// TwinCAT 3 PLC project PLC_1
// ProgramVersion: 3.1.4026.25
// libraries:
//   SPT Base Types, * (Beckhoff Automation LLC)
//   SPT Components, * (Beckhoff Automation LLC)
//   SPT Event Logger, * (Beckhoff Automation LLC)
//   Tc3_PackML_V2, * (Beckhoff Automation GmbH)
//   Tc3_EventLogger, * (Beckhoff Automation GmbH)
//   Tc2_Standard, * (Beckhoff Automation GmbH)
//   Tc2_System, * (Beckhoff Automation GmbH)
// project tree:
//   Library/DUTs/ ST_AbstractLightSource_Command.TcDUT, ST_AbstractLightSource_HMI.TcDUT, ST_AbstractLightSource_Status.TcDUT, ST_AbstractBinaryDrive_Command.TcDUT, ST_AbstractBinaryDrive_Config.TcDUT, ST_AbstractBinaryDrive_Status.TcDUT, ST_AbstractBinaryDrive_HMI.TcDUT, ST_BaseModule_HMI.TcDUT, ST_Sequence_Status.TcDUT, ST_FG_System_Safety.TcDUT, ST_IlluminatedButton_Config.TcDUT, ST_IlluminatedButton_Status.TcDUT, ST_IlluminatedButton_HMI.TcDUT, ST_SafetyDoor_Config.TcDUT, ST_SafetyDoor_Status.TcDUT, ST_SafetyDoor_HMI.TcDUT, ST_SignalTower_Config.TcDUT, ST_SignalTower_Status.TcDUT, ST_SignalTower_HMI.TcDUT, ST_HMI_FG_System.TcDUT, ST_AbstractCamera_Command.TcDUT, ST_AbstractCamera_Status.TcDUT, ST_AbstractCamera_HMI.TcDUT, ST_AbstractBunker_Command.TcDUT, ST_AbstractBunker_Status.TcDUT, ST_AbstractBunker_HMI.TcDUT
//   Library/POUs/ FB_AbstractLightSource.TcPOU, FB_AbstractCamera.TcPOU, FB_AbstractBunker.TcPOU, FB_ControlSource_HMI.TcPOU, FB_ControlSource_Panel.TcPOU, FB_IlluminatedButton.TcPOU, FB_SafetyDoor.TcPOU, FB_SignalTower.TcPOU, FB_AbstractBinaryDrive.TcPOU, F_PMLStateName.TcPOU
//   / PlcTask.TcTTO
//   POUs/ MAIN.TcPOU
//   Modules/00 Machine/ Machine.TcPOU
//   Modules/11 FG_01/ ST_FG_01_Identify_Status.TcDUT, ST_HMI_FG_01.TcDUT, FG_01.TcPOU
//   Modules/12 FG_02/ ST_FG_02_Inspection_Status.TcDUT, ST_HMI_FG_02.TcDUT, FG_02.TcPOU
//   Modules/13 FG_03/ ST_FG_03_Transfer_Status.TcDUT, ST_HMI_FG_03.TcDUT, FG_03.TcPOU
//   Modules/14 FG_04/ ST_FG_04_Press_Status.TcDUT, ST_HMI_FG_04.TcDUT, FG_04.TcPOU
//   Modules/15 FG_05/ ST_FG_05_Capping_Status.TcDUT, ST_HMI_FG_05.TcDUT, FG_05.TcPOU
//   Modules/01 FG_System/ FG_System.TcPOU
//   Modules/10 FG_Transport/ ST_TransferIndex_HMI.TcDUT, ST_TransferIndex_Status.TcDUT, ST_TransferLift_HMI.TcDUT, ST_TransferLift_Status.TcDUT, ST_TransferStopper_HMI.TcDUT, ST_TransferStopper_Status.TcDUT, FG_Transport.TcPOU, FB_TransferIndex.TcPOU, FB_TransferStopper.TcPOU, FB_TransferLift.TcPOU
// (motion and I/O tree: see PLC project sim_1)
// real-time tasks:
//   TASK PlcTask_SIM: cycle T#1ms, priority 4, ADS port 350
//   TASK PlcTask_PLC: cycle T#10ms, priority 20, ADS port 351
// variable links:
//   PLC_1/PLC_1 Instance <-> EtherCAT_1/FG_01_EK1100/FG_01_EL1008_1
//     PlcTask Inputs/MAIN.Machine.FG_01.Y_Gripper.ExtendedSensor <-> Channel 2/Input
//     PlcTask Inputs/MAIN.Machine.FG_01.Y_Gripper.RetractedSensor <-> Channel 1/Input
//     PlcTask Inputs/MAIN.Machine.FG_01.Y_Platform.ExtendedSensor <-> Channel 4/Input
//     PlcTask Inputs/MAIN.Machine.FG_01.Y_Platform.RetractedSensor <-> Channel 3/Input
//     PlcTask Inputs/MAIN.Machine.FG_01.Y_ReaderWindow.ExtendedSensor <-> Channel 6/Input
//     PlcTask Inputs/MAIN.Machine.FG_01.Y_ReaderWindow.RetractedSensor <-> Channel 5/Input
//   PLC_1/PLC_1 Instance <-> EtherCAT_1/FG_01_EK1100/FG_01_EL1008_2
//     PlcTask Inputs/MAIN.Machine.FG_01.B_SafetyGate1.HardwareInput <-> Channel 5/Input
//     PlcTask Inputs/MAIN.Machine.FG_01.B_SafetyGate2.HardwareInput <-> Channel 6/Input
//     PlcTask Inputs/MAIN.Machine.FG_01.Y_Gate1.ExtendedSensor <-> Channel 2/Input
//     PlcTask Inputs/MAIN.Machine.FG_01.Y_Gate2.ExtendedSensor <-> Channel 4/Input
//     PlcTask Inputs/MAIN.Machine.FG_01.Y_Gate1.RetractedSensor <-> Channel 1/Input
//     PlcTask Inputs/MAIN.Machine.FG_01.Y_Gate2.RetractedSensor <-> Channel 3/Input
//   PLC_1/PLC_1 Instance <-> EtherCAT_1/FG_01_EK1100/FG_01_EL1859_1
//     PlcTask Inputs/MAIN.Machine.FG_01.P_Camera.InputData <-> Channel 1/Input
//     PlcTask Inputs/MAIN.Machine.FG_01.P_Camera.InputData @bit 1 <-> Channel 2/Input
//     PlcTask Inputs/MAIN.Machine.FG_01.P_Camera.InputData @bit 2 <-> Channel 3/Input
//     PlcTask Inputs/MAIN.Machine.FG_01.P_Camera.InputData @bit 3 <-> Channel 4/Input
//     PlcTask Inputs/MAIN.Machine.FG_01.P_Camera.InputData @bit 4 <-> Channel 5/Input
//     PlcTask Inputs/MAIN.Machine.FG_01.P_Camera.InputData @bit 5 <-> Channel 6/Input
//     PlcTask Inputs/MAIN.Machine.FG_01.P_Camera.InputData @bit 6 <-> Channel 7/Input
//     PlcTask Inputs/MAIN.Machine.FG_01.P_Camera.InputData @bit 7 <-> Channel 8/Input
//     PlcTask Outputs/MAIN.Machine.FG_01.P_Camera.OutputData @bit 1 <-> Channel 10/Output
//     PlcTask Outputs/MAIN.Machine.FG_01.P_Camera.OutputData @bit 2 <-> Channel 11/Output
//     PlcTask Outputs/MAIN.Machine.FG_01.P_Camera.OutputData @bit 3 <-> Channel 12/Output
//     PlcTask Outputs/MAIN.Machine.FG_01.P_Camera.OutputData @bit 4 <-> Channel 13/Output
//     PlcTask Outputs/MAIN.Machine.FG_01.P_Camera.OutputData @bit 5 <-> Channel 14/Output
//     PlcTask Outputs/MAIN.Machine.FG_01.P_Camera.OutputData @bit 6 <-> Channel 15/Output
//     PlcTask Outputs/MAIN.Machine.FG_01.P_Camera.OutputData @bit 7 <-> Channel 16/Output
//     PlcTask Outputs/MAIN.Machine.FG_01.P_Camera.OutputData <-> Channel 9/Output
//   PLC_1/PLC_1 Instance <-> EtherCAT_1/FG_01_EK1100/FG_01_EL1859_2
//     PlcTask Inputs/MAIN.Machine.FG_01.Y_LaserMark.InputData <-> Channel 1/Input
//     PlcTask Inputs/MAIN.Machine.FG_01.Y_LaserMark.InputData @bit 1 <-> Channel 2/Input
//     PlcTask Inputs/MAIN.Machine.FG_01.Y_LaserMark.InputData @bit 2 <-> Channel 3/Input
//     PlcTask Inputs/MAIN.Machine.FG_01.Y_LaserMark.InputData @bit 3 <-> Channel 4/Input
//     PlcTask Inputs/MAIN.Machine.FG_01.Y_LaserMark.InputData @bit 4 <-> Channel 5/Input
//     PlcTask Inputs/MAIN.Machine.FG_01.Y_LaserMark.InputData @bit 5 <-> Channel 6/Input
//     PlcTask Inputs/MAIN.Machine.FG_01.Y_LaserMark.InputData @bit 6 <-> Channel 7/Input
//     PlcTask Inputs/MAIN.Machine.FG_01.Y_LaserMark.InputData @bit 7 <-> Channel 8/Input
//     PlcTask Outputs/MAIN.Machine.FG_01.Y_LaserMark.OutputData @bit 1 <-> Channel 10/Output
//     PlcTask Outputs/MAIN.Machine.FG_01.Y_LaserMark.OutputData @bit 2 <-> Channel 11/Output
//     PlcTask Outputs/MAIN.Machine.FG_01.Y_LaserMark.OutputData @bit 3 <-> Channel 12/Output
//     PlcTask Outputs/MAIN.Machine.FG_01.Y_LaserMark.OutputData @bit 4 <-> Channel 13/Output
//     PlcTask Outputs/MAIN.Machine.FG_01.Y_LaserMark.OutputData @bit 5 <-> Channel 14/Output
//     PlcTask Outputs/MAIN.Machine.FG_01.Y_LaserMark.OutputData @bit 6 <-> Channel 15/Output
//     PlcTask Outputs/MAIN.Machine.FG_01.Y_LaserMark.OutputData @bit 7 <-> Channel 16/Output
//     PlcTask Outputs/MAIN.Machine.FG_01.Y_LaserMark.OutputData <-> Channel 9/Output
//   PLC_1/PLC_1 Instance <-> EtherCAT_1/FG_01_EK1100/FG_01_EL2008_1
//     PlcTask Outputs/MAIN.Machine.FG_01.Y_Gate1._ExtendOutput <-> Channel 7/Output
//     PlcTask Outputs/MAIN.Machine.FG_01.Y_Gate2._ExtendOutput <-> Channel 8/Output
//     PlcTask Outputs/MAIN.Machine.FG_01.Y_Gripper._ExtendOutput <-> Channel 1/Output
//     PlcTask Outputs/MAIN.Machine.FG_01.Y_Gripper._RetractOutput <-> Channel 5/Output
//     PlcTask Outputs/MAIN.Machine.FG_01.Y_Platform._ExtendOutput <-> Channel 2/Output
//     PlcTask Outputs/MAIN.Machine.FG_01.Y_Platform._RetractOutput <-> Channel 3/Output
//     PlcTask Outputs/MAIN.Machine.FG_01.Y_ReaderWindow._ExtendOutput <-> Channel 4/Output
//     PlcTask Outputs/MAIN.Machine.FG_01.Y_ReaderWindow._RetractOutput <-> Channel 6/Output
//   PLC_1/PLC_1 Instance <-> EtherCAT_1/FG_02_EK1100/FG_02_EL1859_1
//     PlcTask Inputs/MAIN.Machine.FG_02.P_Camera.InputData <-> Channel 1/Input
//     PlcTask Inputs/MAIN.Machine.FG_02.P_Camera.InputData @bit 1 <-> Channel 2/Input
//     PlcTask Inputs/MAIN.Machine.FG_02.P_Camera.InputData @bit 2 <-> Channel 3/Input
//     PlcTask Inputs/MAIN.Machine.FG_02.P_Camera.InputData @bit 3 <-> Channel 4/Input
//     PlcTask Inputs/MAIN.Machine.FG_02.P_Camera.InputData @bit 4 <-> Channel 5/Input
//     PlcTask Inputs/MAIN.Machine.FG_02.P_Camera.InputData @bit 5 <-> Channel 6/Input
//     PlcTask Inputs/MAIN.Machine.FG_02.P_Camera.InputData @bit 6 <-> Channel 7/Input
//     PlcTask Inputs/MAIN.Machine.FG_02.P_Camera.InputData @bit 7 <-> Channel 8/Input
//     PlcTask Outputs/MAIN.Machine.FG_02.P_Camera.OutputData @bit 1 <-> Channel 10/Output
//     PlcTask Outputs/MAIN.Machine.FG_02.P_Camera.OutputData @bit 2 <-> Channel 11/Output
//     PlcTask Outputs/MAIN.Machine.FG_02.P_Camera.OutputData @bit 3 <-> Channel 12/Output
//     PlcTask Outputs/MAIN.Machine.FG_02.P_Camera.OutputData @bit 4 <-> Channel 13/Output
//     PlcTask Outputs/MAIN.Machine.FG_02.P_Camera.OutputData @bit 5 <-> Channel 14/Output
//     PlcTask Outputs/MAIN.Machine.FG_02.P_Camera.OutputData @bit 6 <-> Channel 15/Output
//     PlcTask Outputs/MAIN.Machine.FG_02.P_Camera.OutputData @bit 7 <-> Channel 16/Output
//     PlcTask Outputs/MAIN.Machine.FG_02.P_Camera.OutputData <-> Channel 9/Output
//   PLC_1/PLC_1 Instance <-> EtherCAT_1/FG_03_EK1100/FG_03_EL1809_1
//     PlcTask Inputs/MAIN.Machine.FG_03.B_Detect1.HardwareInput <-> Channel 15/Input
//     PlcTask Inputs/MAIN.Machine.FG_03.B_Detect2.HardwareInput <-> Channel 16/Input
//     PlcTask Inputs/MAIN.Machine.FG_03.Y_AxisR1.ExtendedSensor <-> Channel 5/Input
//     PlcTask Inputs/MAIN.Machine.FG_03.Y_AxisR1.RetractedSensor <-> Channel 6/Input
//     PlcTask Inputs/MAIN.Machine.FG_03.Y_AxisX1.ExtendedSensor <-> Channel 1/Input
//     PlcTask Inputs/MAIN.Machine.FG_03.Y_AxisX2.ExtendedSensor <-> Channel 9/Input
//     PlcTask Inputs/MAIN.Machine.FG_03.Y_AxisX1.RetractedSensor <-> Channel 2/Input
//     PlcTask Inputs/MAIN.Machine.FG_03.Y_AxisX2.RetractedSensor <-> Channel 10/Input
//     PlcTask Inputs/MAIN.Machine.FG_03.Y_AxisY1.ExtendedSensor <-> Channel 3/Input
//     PlcTask Inputs/MAIN.Machine.FG_03.Y_AxisY2.ExtendedSensor <-> Channel 11/Input
//     PlcTask Inputs/MAIN.Machine.FG_03.Y_AxisY1.RetractedSensor <-> Channel 4/Input
//     PlcTask Inputs/MAIN.Machine.FG_03.Y_AxisY2.RetractedSensor <-> Channel 12/Input
//     PlcTask Inputs/MAIN.Machine.FG_03.Y_Gripper1.ExtendedSensor <-> Channel 7/Input
//     PlcTask Inputs/MAIN.Machine.FG_03.Y_Gripper2.ExtendedSensor <-> Channel 13/Input
//     PlcTask Inputs/MAIN.Machine.FG_03.Y_Gripper1.RetractedSensor <-> Channel 8/Input
//     PlcTask Inputs/MAIN.Machine.FG_03.Y_Gripper2.RetractedSensor <-> Channel 14/Input
//   PLC_1/PLC_1 Instance <-> EtherCAT_1/FG_03_EK1100/FG_03_EL2809_1
//     PlcTask Outputs/MAIN.Machine.FG_03.Y_AxisR1._ExtendOutput <-> Channel 5/Output
//     PlcTask Outputs/MAIN.Machine.FG_03.Y_AxisR1._RetractOutput <-> Channel 6/Output
//     PlcTask Outputs/MAIN.Machine.FG_03.Y_AxisX1._ExtendOutput <-> Channel 1/Output
//     PlcTask Outputs/MAIN.Machine.FG_03.Y_AxisX2._ExtendOutput <-> Channel 9/Output
//     PlcTask Outputs/MAIN.Machine.FG_03.Y_AxisX1._RetractOutput <-> Channel 2/Output
//     PlcTask Outputs/MAIN.Machine.FG_03.Y_AxisX2._RetractOutput <-> Channel 10/Output
//     PlcTask Outputs/MAIN.Machine.FG_03.Y_AxisY1._ExtendOutput <-> Channel 3/Output
//     PlcTask Outputs/MAIN.Machine.FG_03.Y_AxisY2._ExtendOutput <-> Channel 11/Output
//     PlcTask Outputs/MAIN.Machine.FG_03.Y_AxisY1._RetractOutput <-> Channel 4/Output
//     PlcTask Outputs/MAIN.Machine.FG_03.Y_AxisY2._RetractOutput <-> Channel 12/Output
//     PlcTask Outputs/MAIN.Machine.FG_03.Y_Gripper1._ExtendOutput <-> Channel 7/Output
//     PlcTask Outputs/MAIN.Machine.FG_03.Y_Gripper2._ExtendOutput <-> Channel 13/Output
//     PlcTask Outputs/MAIN.Machine.FG_03.Y_Gripper1._RetractOutput <-> Channel 8/Output
//     PlcTask Outputs/MAIN.Machine.FG_03.Y_Gripper2._RetractOutput <-> Channel 14/Output
//   PLC_1/PLC_1 Instance <-> EtherCAT_1/FG_04_EK1100/FG_04_EL1008_1
//     PlcTask Inputs/MAIN.Machine.FG_04.B_NIO.HardwareInput <-> Channel 3/Input
//     PlcTask Inputs/MAIN.Machine.FG_04.Y_AxisZ.ExtendedSensor <-> Channel 1/Input
//     PlcTask Inputs/MAIN.Machine.FG_04.Y_AxisZ.RetractedSensor <-> Channel 2/Input
//   PLC_1/PLC_1 Instance <-> EtherCAT_1/FG_04_EK1100/FG_04_EL2008_1
//     PlcTask Outputs/MAIN.Machine.FG_04.Y_AxisZ._ExtendOutput <-> Channel 1/Output
//     PlcTask Outputs/MAIN.Machine.FG_04.Y_AxisZ._RetractOutput <-> Channel 2/Output
//   PLC_1/PLC_1 Instance <-> EtherCAT_1/FG_05_EK1100/FG_05_EL1809_1
//     PlcTask Inputs/MAIN.Machine.FG_05.B_Detect.HardwareInput <-> Channel 14/Input
//     PlcTask Inputs/MAIN.Machine.FG_05.B_Part.HardwareInput <-> Channel 13/Input
//     PlcTask Inputs/MAIN.Machine.FG_05.Y_AxisR.ExtendedSensor <-> Channel 7/Input
//     PlcTask Inputs/MAIN.Machine.FG_05.Y_AxisR.RetractedSensor <-> Channel 8/Input
//     PlcTask Inputs/MAIN.Machine.FG_05.Y_AxisX.ExtendedSensor <-> Channel 1/Input
//     PlcTask Inputs/MAIN.Machine.FG_05.Y_AxisX.RetractedSensor <-> Channel 2/Input
//     PlcTask Inputs/MAIN.Machine.FG_05.Y_AxisZ1.ExtendedSensor <-> Channel 3/Input
//     PlcTask Inputs/MAIN.Machine.FG_05.Y_AxisZ2.ExtendedSensor <-> Channel 5/Input
//     PlcTask Inputs/MAIN.Machine.FG_05.Y_AxisZ1.RetractedSensor <-> Channel 4/Input
//     PlcTask Inputs/MAIN.Machine.FG_05.Y_AxisZ2.RetractedSensor <-> Channel 6/Input
//     PlcTask Inputs/MAIN.Machine.FG_05.Y_CapsSourceStopper.ExtendedSensor <-> Channel 11/Input
//     PlcTask Inputs/MAIN.Machine.FG_05.Y_CapsSourceStopper.RetractedSensor <-> Channel 12/Input
//     PlcTask Inputs/MAIN.Machine.FG_05.Y_Gripper.ExtendedSensor <-> Channel 9/Input
//     PlcTask Inputs/MAIN.Machine.FG_05.Y_Gripper.RetractedSensor <-> Channel 10/Input
//   PLC_1/PLC_1 Instance <-> EtherCAT_1/FG_05_EK1100/FG_05_EL1859_1
//     PlcTask Inputs/MAIN.Machine.FG_05.Y_CapsSource.InputData <-> Channel 1/Input
//     PlcTask Inputs/MAIN.Machine.FG_05.Y_CapsSource.InputData @bit 1 <-> Channel 2/Input
//     PlcTask Inputs/MAIN.Machine.FG_05.Y_CapsSource.InputData @bit 2 <-> Channel 3/Input
//     PlcTask Inputs/MAIN.Machine.FG_05.Y_CapsSource.InputData @bit 3 <-> Channel 4/Input
//     PlcTask Inputs/MAIN.Machine.FG_05.Y_CapsSource.InputData @bit 4 <-> Channel 5/Input
//     PlcTask Inputs/MAIN.Machine.FG_05.Y_CapsSource.InputData @bit 5 <-> Channel 6/Input
//     PlcTask Inputs/MAIN.Machine.FG_05.Y_CapsSource.InputData @bit 6 <-> Channel 7/Input
//     PlcTask Inputs/MAIN.Machine.FG_05.Y_CapsSource.InputData @bit 7 <-> Channel 8/Input
//     PlcTask Outputs/MAIN.Machine.FG_05.Y_CapsSource.OutputData @bit 1 <-> Channel 10/Output
//     PlcTask Outputs/MAIN.Machine.FG_05.Y_CapsSource.OutputData @bit 2 <-> Channel 11/Output
//     PlcTask Outputs/MAIN.Machine.FG_05.Y_CapsSource.OutputData @bit 3 <-> Channel 12/Output
//     PlcTask Outputs/MAIN.Machine.FG_05.Y_CapsSource.OutputData @bit 4 <-> Channel 13/Output
//     PlcTask Outputs/MAIN.Machine.FG_05.Y_CapsSource.OutputData @bit 5 <-> Channel 14/Output
//     PlcTask Outputs/MAIN.Machine.FG_05.Y_CapsSource.OutputData @bit 6 <-> Channel 15/Output
//     PlcTask Outputs/MAIN.Machine.FG_05.Y_CapsSource.OutputData @bit 7 <-> Channel 16/Output
//     PlcTask Outputs/MAIN.Machine.FG_05.Y_CapsSource.OutputData <-> Channel 9/Output
//   PLC_1/PLC_1 Instance <-> EtherCAT_1/FG_05_EK1100/FG_05_EL1859_2
//     PlcTask Inputs/MAIN.Machine.FG_05.P_Camera.InputData <-> Channel 1/Input
//     PlcTask Inputs/MAIN.Machine.FG_05.P_Camera.InputData @bit 1 <-> Channel 2/Input
//     PlcTask Inputs/MAIN.Machine.FG_05.P_Camera.InputData @bit 2 <-> Channel 3/Input
//     PlcTask Inputs/MAIN.Machine.FG_05.P_Camera.InputData @bit 3 <-> Channel 4/Input
//     PlcTask Inputs/MAIN.Machine.FG_05.P_Camera.InputData @bit 4 <-> Channel 5/Input
//     PlcTask Inputs/MAIN.Machine.FG_05.P_Camera.InputData @bit 5 <-> Channel 6/Input
//     PlcTask Inputs/MAIN.Machine.FG_05.P_Camera.InputData @bit 6 <-> Channel 7/Input
//     PlcTask Inputs/MAIN.Machine.FG_05.P_Camera.InputData @bit 7 <-> Channel 8/Input
//     PlcTask Outputs/MAIN.Machine.FG_05.P_Camera.OutputData @bit 1 <-> Channel 10/Output
//     PlcTask Outputs/MAIN.Machine.FG_05.P_Camera.OutputData @bit 2 <-> Channel 11/Output
//     PlcTask Outputs/MAIN.Machine.FG_05.P_Camera.OutputData @bit 3 <-> Channel 12/Output
//     PlcTask Outputs/MAIN.Machine.FG_05.P_Camera.OutputData @bit 4 <-> Channel 13/Output
//     PlcTask Outputs/MAIN.Machine.FG_05.P_Camera.OutputData @bit 5 <-> Channel 14/Output
//     PlcTask Outputs/MAIN.Machine.FG_05.P_Camera.OutputData @bit 6 <-> Channel 15/Output
//     PlcTask Outputs/MAIN.Machine.FG_05.P_Camera.OutputData @bit 7 <-> Channel 16/Output
//     PlcTask Outputs/MAIN.Machine.FG_05.P_Camera.OutputData <-> Channel 9/Output
//   PLC_1/PLC_1 Instance <-> EtherCAT_1/FG_05_EK1100/FG_05_EL2809_1
//     PlcTask Outputs/MAIN.Machine.FG_05.Y_AxisR._ExtendOutput <-> Channel 7/Output
//     PlcTask Outputs/MAIN.Machine.FG_05.Y_AxisR._RetractOutput <-> Channel 8/Output
//     PlcTask Outputs/MAIN.Machine.FG_05.Y_AxisX._ExtendOutput <-> Channel 1/Output
//     PlcTask Outputs/MAIN.Machine.FG_05.Y_AxisX._RetractOutput <-> Channel 2/Output
//     PlcTask Outputs/MAIN.Machine.FG_05.Y_AxisZ1._ExtendOutput <-> Channel 3/Output
//     PlcTask Outputs/MAIN.Machine.FG_05.Y_AxisZ2._ExtendOutput <-> Channel 5/Output
//     PlcTask Outputs/MAIN.Machine.FG_05.Y_AxisZ1._RetractOutput <-> Channel 4/Output
//     PlcTask Outputs/MAIN.Machine.FG_05.Y_AxisZ2._RetractOutput <-> Channel 6/Output
//     PlcTask Outputs/MAIN.Machine.FG_05.Y_CapsSourceStopper._ExtendOutput <-> Channel 11/Output
//     PlcTask Outputs/MAIN.Machine.FG_05.Y_CapsSourceStopper._RetractOutput <-> Channel 12/Output
//     PlcTask Outputs/MAIN.Machine.FG_05.Y_Gripper._ExtendOutput <-> Channel 9/Output
//     PlcTask Outputs/MAIN.Machine.FG_05.Y_Gripper._RetractOutput <-> Channel 10/Output
//   PLC_1/PLC_1 Instance <-> EtherCAT_1/FG_System_EK1100/FG_System_Door_EL1809_1
//     PlcTask Inputs/MAIN.Machine.FG_System.B_SafetyDoor11.ClosedSensor <-> Channel 1/Input
//     PlcTask Inputs/MAIN.Machine.FG_System.B_SafetyDoor12.ClosedSensor <-> Channel 3/Input
//     PlcTask Inputs/MAIN.Machine.FG_System.B_SafetyDoor13.ClosedSensor <-> Channel 5/Input
//     PlcTask Inputs/MAIN.Machine.FG_System.B_SafetyDoor21.ClosedSensor <-> Channel 7/Input
//     PlcTask Inputs/MAIN.Machine.FG_System.B_SafetyDoor22.ClosedSensor <-> Channel 9/Input
//     PlcTask Inputs/MAIN.Machine.FG_System.B_SafetyDoor23.ClosedSensor <-> Channel 11/Input
//     PlcTask Inputs/MAIN.Machine.FG_System.B_SafetyDoor11.LockedSensor <-> Channel 2/Input
//     PlcTask Inputs/MAIN.Machine.FG_System.B_SafetyDoor12.LockedSensor <-> Channel 4/Input
//     PlcTask Inputs/MAIN.Machine.FG_System.B_SafetyDoor13.LockedSensor <-> Channel 6/Input
//     PlcTask Inputs/MAIN.Machine.FG_System.B_SafetyDoor21.LockedSensor <-> Channel 8/Input
//     PlcTask Inputs/MAIN.Machine.FG_System.B_SafetyDoor22.LockedSensor <-> Channel 10/Input
//     PlcTask Inputs/MAIN.Machine.FG_System.B_SafetyDoor23.LockedSensor <-> Channel 12/Input
//   PLC_1/PLC_1 Instance <-> EtherCAT_1/FG_System_EK1100/FG_System_Door_EL2008_1
//     PlcTask Outputs/MAIN.Machine.FG_System.B_SafetyDoor11.LockOutput <-> Channel 1/Output
//     PlcTask Outputs/MAIN.Machine.FG_System.B_SafetyDoor12.LockOutput <-> Channel 2/Output
//     PlcTask Outputs/MAIN.Machine.FG_System.B_SafetyDoor13.LockOutput <-> Channel 3/Output
//     PlcTask Outputs/MAIN.Machine.FG_System.B_SafetyDoor21.LockOutput <-> Channel 4/Output
//     PlcTask Outputs/MAIN.Machine.FG_System.B_SafetyDoor22.LockOutput <-> Channel 5/Output
//     PlcTask Outputs/MAIN.Machine.FG_System.B_SafetyDoor23.LockOutput <-> Channel 6/Output
//   PLC_1/PLC_1 Instance <-> EtherCAT_1/FG_System_EK1100/FG_System_Panel_EL1809_1
//     PlcTask Inputs/MAIN.ControlSource_Panel.AbortPressed <-> Channel 5/Input
//     PlcTask Inputs/MAIN.ControlSource_Panel.ClearPressed <-> Channel 4/Input
//     PlcTask Inputs/MAIN.ControlSource_Panel.MainPMLControl_Simplified.ResetPressed <-> Channel 2/Input
//     PlcTask Inputs/MAIN.ControlSource_Panel.MainPMLControl_Simplified.StartPressed <-> Channel 1/Input
//     PlcTask Inputs/MAIN.ControlSource_Panel.MainPMLControl_Simplified.StopPressed <-> Channel 3/Input
//     PlcTask Inputs/MAIN.ControlSource_Panel.MaintenancePressed <-> Channel 7/Input
//     PlcTask Inputs/MAIN.ControlSource_Panel.ManualPressed <-> Channel 8/Input
//     PlcTask Inputs/MAIN.ControlSource_Panel.ProductionPressed <-> Channel 6/Input
//     PlcTask Inputs/MAIN.Machine.FG_System.SS_EStop1.HardwareInput <-> Channel 9/Input
//     PlcTask Inputs/MAIN.Machine.FG_System.SS_EStop2.HardwareInput <-> Channel 10/Input
//   PLC_1/PLC_1 Instance <-> EtherCAT_1/FG_System_EK1100/FG_System_Panel_EL2809_1
//     PlcTask Outputs/MAIN.ControlSource_Panel.LampAbort <-> Channel 5/Output
//     PlcTask Outputs/MAIN.ControlSource_Panel.LampClear <-> Channel 4/Output
//     PlcTask Outputs/MAIN.ControlSource_Panel.LampMaintenance <-> Channel 7/Output
//     PlcTask Outputs/MAIN.ControlSource_Panel.LampManual <-> Channel 8/Output
//     PlcTask Outputs/MAIN.ControlSource_Panel.LampProduction <-> Channel 6/Output
//     PlcTask Outputs/MAIN.ControlSource_Panel.LampReset <-> Channel 2/Output
//     PlcTask Outputs/MAIN.ControlSource_Panel.LampStart <-> Channel 1/Output
//     PlcTask Outputs/MAIN.ControlSource_Panel.LampStop <-> Channel 3/Output
//     PlcTask Outputs/MAIN.Machine.FG_System.H_SignalTower.Blue <-> Channel 11/Output
//     PlcTask Outputs/MAIN.Machine.FG_System.H_SignalTower.Green <-> Channel 12/Output
//     PlcTask Outputs/MAIN.Machine.FG_System.H_SignalTower.Red <-> Channel 9/Output
//     PlcTask Outputs/MAIN.Machine.FG_System.H_SignalTower.Yellow <-> Channel 10/Output
//     PlcTask Outputs/MAIN.Machine.FG_System.SS_EStop1.LampOutput <-> Channel 13/Output
//     PlcTask Outputs/MAIN.Machine.FG_System.SS_EStop2.LampOutput <-> Channel 14/Output
//   PLC_1/PLC_1 Instance <-> EtherCAT_1/FG_Transport_EK1100/FG_Transport_Drive_EL1008_1
//     PlcTask Inputs/MAIN.Machine.FG_Transport.Transport01._DriveActive <-> Channel 1/Input
//     PlcTask Inputs/MAIN.Machine.FG_Transport.Transport02._DriveActive <-> Channel 2/Input
//   PLC_1/PLC_1 Instance <-> EtherCAT_1/FG_Transport_EK1100/FG_Transport_Drive_EL2008_1
//     PlcTask Outputs/MAIN.Machine.FG_Transport.Transport01._Backward <-> Channel 1/Output
//     PlcTask Outputs/MAIN.Machine.FG_Transport.Transport02._Backward <-> Channel 3/Output
//     PlcTask Outputs/MAIN.Machine.FG_Transport.Transport01._Forward <-> Channel 2/Output
//     PlcTask Outputs/MAIN.Machine.FG_Transport.Transport02._Forward <-> Channel 4/Output
//   PLC_1/PLC_1 Instance <-> EtherCAT_1/FG_Transport_EK1100/FG_Transport_Index_EL1809_1
//     PlcTask Inputs/MAIN.Machine.FG_Transport.Index01.B_Detect.HardwareInput <-> Channel 1/Input
//     PlcTask Inputs/MAIN.Machine.FG_Transport.Index02.B_Detect.HardwareInput <-> Channel 7/Input
//     PlcTask Inputs/MAIN.Machine.FG_Transport.Index03.B_Detect.HardwareInput <-> Channel 13/Input
//     PlcTask Inputs/MAIN.Machine.FG_Transport.Index01.B_Exit.HardwareInput <-> Channel 2/Input
//     PlcTask Inputs/MAIN.Machine.FG_Transport.Index02.B_Exit.HardwareInput <-> Channel 8/Input
//     PlcTask Inputs/MAIN.Machine.FG_Transport.Index03.B_Exit.HardwareInput <-> Channel 14/Input
//     PlcTask Inputs/MAIN.Machine.FG_Transport.Index01.Y_Lift.ExtendedSensor <-> Channel 4/Input
//     PlcTask Inputs/MAIN.Machine.FG_Transport.Index02.Y_Lift.ExtendedSensor <-> Channel 10/Input
//     PlcTask Inputs/MAIN.Machine.FG_Transport.Index03.Y_Lift.ExtendedSensor <-> Channel 16/Input
//     PlcTask Inputs/MAIN.Machine.FG_Transport.Index01.Y_Lift.RetractedSensor <-> Channel 3/Input
//     PlcTask Inputs/MAIN.Machine.FG_Transport.Index02.Y_Lift.RetractedSensor <-> Channel 9/Input
//     PlcTask Inputs/MAIN.Machine.FG_Transport.Index03.Y_Lift.RetractedSensor <-> Channel 15/Input
//     PlcTask Inputs/MAIN.Machine.FG_Transport.Index01.Y_Stopper.ExtendedSensor <-> Channel 6/Input
//     PlcTask Inputs/MAIN.Machine.FG_Transport.Index02.Y_Stopper.ExtendedSensor <-> Channel 12/Input
//     PlcTask Inputs/MAIN.Machine.FG_Transport.Index01.Y_Stopper.RetractedSensor <-> Channel 5/Input
//     PlcTask Inputs/MAIN.Machine.FG_Transport.Index02.Y_Stopper.RetractedSensor <-> Channel 11/Input
//   PLC_1/PLC_1 Instance <-> EtherCAT_1/FG_Transport_EK1100/FG_Transport_Index_EL1809_2
//     PlcTask Inputs/MAIN.Machine.FG_Transport.Index03.Y_Stopper.ExtendedSensor <-> Channel 2/Input
//     PlcTask Inputs/MAIN.Machine.FG_Transport.Index04.Y_Stopper.ExtendedSensor <-> Channel 8/Input
//     PlcTask Inputs/MAIN.Machine.FG_Transport.Index05.Y_Stopper.ExtendedSensor <-> Channel 14/Input
//     PlcTask Inputs/MAIN.Machine.FG_Transport.Index03.Y_Stopper.RetractedSensor <-> Channel 1/Input
//     PlcTask Inputs/MAIN.Machine.FG_Transport.Index04.Y_Stopper.RetractedSensor <-> Channel 7/Input
//     PlcTask Inputs/MAIN.Machine.FG_Transport.Index05.Y_Stopper.RetractedSensor <-> Channel 13/Input
//     PlcTask Inputs/MAIN.Machine.FG_Transport.Index04.B_Detect.HardwareInput <-> Channel 3/Input
//     PlcTask Inputs/MAIN.Machine.FG_Transport.Index05.B_Detect.HardwareInput <-> Channel 9/Input
//     PlcTask Inputs/MAIN.Machine.FG_Transport.Index04.B_Exit.HardwareInput <-> Channel 4/Input
//     PlcTask Inputs/MAIN.Machine.FG_Transport.Index05.B_Exit.HardwareInput <-> Channel 10/Input
//     PlcTask Inputs/MAIN.Machine.FG_Transport.Index04.Y_Lift.ExtendedSensor <-> Channel 6/Input
//     PlcTask Inputs/MAIN.Machine.FG_Transport.Index05.Y_Lift.ExtendedSensor <-> Channel 12/Input
//     PlcTask Inputs/MAIN.Machine.FG_Transport.Index04.Y_Lift.RetractedSensor <-> Channel 5/Input
//     PlcTask Inputs/MAIN.Machine.FG_Transport.Index05.Y_Lift.RetractedSensor <-> Channel 11/Input
//   PLC_1/PLC_1 Instance <-> EtherCAT_1/FG_Transport_EK1100/FG_Transport_Index_EL2809_1
//     PlcTask Outputs/MAIN.Machine.FG_Transport.Index01.Y_Lift._ExtendOutput <-> Channel 2/Output
//     PlcTask Outputs/MAIN.Machine.FG_Transport.Index02.Y_Lift._ExtendOutput <-> Channel 5/Output
//     PlcTask Outputs/MAIN.Machine.FG_Transport.Index03.Y_Lift._ExtendOutput <-> Channel 8/Output
//     PlcTask Outputs/MAIN.Machine.FG_Transport.Index04.Y_Lift._ExtendOutput <-> Channel 11/Output
//     PlcTask Outputs/MAIN.Machine.FG_Transport.Index05.Y_Lift._ExtendOutput <-> Channel 14/Output
//     PlcTask Outputs/MAIN.Machine.FG_Transport.Index01.Y_Lift._RetractOutput <-> Channel 1/Output
//     PlcTask Outputs/MAIN.Machine.FG_Transport.Index02.Y_Lift._RetractOutput <-> Channel 4/Output
//     PlcTask Outputs/MAIN.Machine.FG_Transport.Index03.Y_Lift._RetractOutput <-> Channel 7/Output
//     PlcTask Outputs/MAIN.Machine.FG_Transport.Index04.Y_Lift._RetractOutput <-> Channel 10/Output
//     PlcTask Outputs/MAIN.Machine.FG_Transport.Index05.Y_Lift._RetractOutput <-> Channel 13/Output
//     PlcTask Outputs/MAIN.Machine.FG_Transport.Index01.Y_Stopper._ExtendOutput <-> Channel 3/Output
//     PlcTask Outputs/MAIN.Machine.FG_Transport.Index02.Y_Stopper._ExtendOutput <-> Channel 6/Output
//     PlcTask Outputs/MAIN.Machine.FG_Transport.Index03.Y_Stopper._ExtendOutput <-> Channel 9/Output
//     PlcTask Outputs/MAIN.Machine.FG_Transport.Index04.Y_Stopper._ExtendOutput <-> Channel 12/Output
//     PlcTask Outputs/MAIN.Machine.FG_Transport.Index05.Y_Stopper._ExtendOutput <-> Channel 15/Output
//   PLC_1/PLC_1 Instance <-> EtherCAT_1/FG_Transport_EK1100/FG_Transport_Lift_EL1809_1
//     PlcTask Inputs/MAIN.Machine.FG_Transport.Lift01.B_Detect.HardwareInput <-> Channel 1/Input
//     PlcTask Inputs/MAIN.Machine.FG_Transport.Lift02.B_Detect.HardwareInput <-> Channel 6/Input
//     PlcTask Inputs/MAIN.Machine.FG_Transport.Lift01.B_Exit.HardwareInput <-> Channel 2/Input
//     PlcTask Inputs/MAIN.Machine.FG_Transport.Lift02.B_Exit.HardwareInput <-> Channel 7/Input
//     PlcTask Inputs/MAIN.Machine.FG_Transport.Lift01.M_Conveyor._DriveActive <-> Channel 5/Input
//     PlcTask Inputs/MAIN.Machine.FG_Transport.Lift02.M_Conveyor._DriveActive <-> Channel 10/Input
//     PlcTask Inputs/MAIN.Machine.FG_Transport.Lift01.Y_Lift.ExtendedSensor <-> Channel 4/Input
//     PlcTask Inputs/MAIN.Machine.FG_Transport.Lift02.Y_Lift.ExtendedSensor <-> Channel 9/Input
//     PlcTask Inputs/MAIN.Machine.FG_Transport.Lift01.Y_Lift.RetractedSensor <-> Channel 3/Input
//     PlcTask Inputs/MAIN.Machine.FG_Transport.Lift02.Y_Lift.RetractedSensor <-> Channel 8/Input
//   PLC_1/PLC_1 Instance <-> EtherCAT_1/FG_Transport_EK1100/FG_Transport_Lift_EL2008_1
//     PlcTask Outputs/MAIN.Machine.FG_Transport.Lift01.M_Conveyor._Backward <-> Channel 3/Output
//     PlcTask Outputs/MAIN.Machine.FG_Transport.Lift02.M_Conveyor._Backward <-> Channel 7/Output
//     PlcTask Outputs/MAIN.Machine.FG_Transport.Lift01.M_Conveyor._Forward <-> Channel 4/Output
//     PlcTask Outputs/MAIN.Machine.FG_Transport.Lift02.M_Conveyor._Forward <-> Channel 8/Output
//     PlcTask Outputs/MAIN.Machine.FG_Transport.Lift01.Y_Lift._ExtendOutput <-> Channel 2/Output
//     PlcTask Outputs/MAIN.Machine.FG_Transport.Lift02.Y_Lift._ExtendOutput <-> Channel 6/Output
//     PlcTask Outputs/MAIN.Machine.FG_Transport.Lift01.Y_Lift._RetractOutput <-> Channel 1/Output
//     PlcTask Outputs/MAIN.Machine.FG_Transport.Lift02.Y_Lift._RetractOutput <-> Channel 5/Output
//   PLC_1/PLC_1 Instance <-> EtherCAT_1/FG_Transport_EK1100/FG_Transport_Stopper_EL1809_1
//     PlcTask Inputs/MAIN.Machine.FG_Transport.Stopper01.B_Detect.HardwareInput <-> Channel 1/Input
//     PlcTask Inputs/MAIN.Machine.FG_Transport.Stopper02.B_Detect.HardwareInput <-> Channel 5/Input
//     PlcTask Inputs/MAIN.Machine.FG_Transport.Stopper03.B_Detect.HardwareInput <-> Channel 9/Input
//     PlcTask Inputs/MAIN.Machine.FG_Transport.Stopper04.B_Detect.HardwareInput <-> Channel 13/Input
//     PlcTask Inputs/MAIN.Machine.FG_Transport.Stopper01.B_Exit.HardwareInput <-> Channel 2/Input
//     PlcTask Inputs/MAIN.Machine.FG_Transport.Stopper02.B_Exit.HardwareInput <-> Channel 6/Input
//     PlcTask Inputs/MAIN.Machine.FG_Transport.Stopper03.B_Exit.HardwareInput <-> Channel 10/Input
//     PlcTask Inputs/MAIN.Machine.FG_Transport.Stopper04.B_Exit.HardwareInput <-> Channel 14/Input
//     PlcTask Inputs/MAIN.Machine.FG_Transport.Stopper01.Y_Stopper.ExtendedSensor <-> Channel 4/Input
//     PlcTask Inputs/MAIN.Machine.FG_Transport.Stopper02.Y_Stopper.ExtendedSensor <-> Channel 8/Input
//     PlcTask Inputs/MAIN.Machine.FG_Transport.Stopper03.Y_Stopper.ExtendedSensor <-> Channel 12/Input
//     PlcTask Inputs/MAIN.Machine.FG_Transport.Stopper04.Y_Stopper.ExtendedSensor <-> Channel 16/Input
//     PlcTask Inputs/MAIN.Machine.FG_Transport.Stopper01.Y_Stopper.RetractedSensor <-> Channel 3/Input
//     PlcTask Inputs/MAIN.Machine.FG_Transport.Stopper02.Y_Stopper.RetractedSensor <-> Channel 7/Input
//     PlcTask Inputs/MAIN.Machine.FG_Transport.Stopper03.Y_Stopper.RetractedSensor <-> Channel 11/Input
//     PlcTask Inputs/MAIN.Machine.FG_Transport.Stopper04.Y_Stopper.RetractedSensor <-> Channel 15/Input
//   PLC_1/PLC_1 Instance <-> EtherCAT_1/FG_Transport_EK1100/FG_Transport_Stopper_EL2008_1
//     PlcTask Outputs/MAIN.Machine.FG_Transport.Stopper01.Y_Stopper._ExtendOutput <-> Channel 1/Output
//     PlcTask Outputs/MAIN.Machine.FG_Transport.Stopper02.Y_Stopper._ExtendOutput <-> Channel 2/Output
//     PlcTask Outputs/MAIN.Machine.FG_Transport.Stopper03.Y_Stopper._ExtendOutput <-> Channel 3/Output
//     PlcTask Outputs/MAIN.Machine.FG_Transport.Stopper04.Y_Stopper._ExtendOutput <-> Channel 4/Output

CONFIGURATION PLC_1
    RESOURCE PLC ON TwinCAT3
        TASK PlcTask(INTERVAL := T#10ms, PRIORITY := 20);
        PROGRAM MAIN WITH PlcTask : MAIN;
    END_RESOURCE
END_CONFIGURATION

// ---- Library/DUTs/ST_AbstractLightSource_Command.TcDUT
TYPE ST_AbstractLightSource_Command :
STRUCT
	Enable : BOOL;
END_STRUCT
END_TYPE

// ---- Library/DUTs/ST_AbstractLightSource_HMI.TcDUT
// Light source HMI interface - ONE struct per tile.
// Extends ST_ComponentBase_HMI, so one bound parameter also carries Config,
// Command and Status - and the added members may not reuse those three names.
TYPE ST_AbstractLightSource_HMI EXTENDS ST_ComponentBase_HMI :
STRUCT
	DeviceCommand	: ST_AbstractLightSource_Command;
	Device			: ST_AbstractLightSource_Status;
END_STRUCT
END_TYPE

// ---- Library/DUTs/ST_AbstractLightSource_Status.TcDUT
TYPE ST_AbstractLightSource_Status :
STRUCT
	Enabled   : BOOL;
	Error     : BOOL;
	ErrorCode : BYTE;
END_STRUCT
END_TYPE

// ---- Library/DUTs/ST_AbstractBinaryDrive_Command.TcDUT
// Honoured by FB_AbstractBinaryDrive itself, in Manual and Maintenance mode only.
// A drive is a bare two direction contactor with no SPT component to jog it
// through, so the command lives here and the block reads its own struct.
// Reached as HMI.DeviceCommand - Command is inherited and therefore taken.
// Both directions are offered: a lift's carriage belt is driven both ways by hand.
// Asking for both at once is a stop, not a fault - CyclicLogic cancels them.
TYPE ST_AbstractBinaryDrive_Command :
STRUCT
	RunForward		: BOOL;
	RunBackward		: BOOL;
END_STRUCT
END_TYPE

// ---- Library/DUTs/ST_AbstractBinaryDrive_Config.TcDUT
TYPE ST_AbstractBinaryDrive_Config :
STRUCT
	StartTime : TIME;
END_STRUCT
END_TYPE

// ---- Library/DUTs/ST_AbstractBinaryDrive_Status.TcDUT
TYPE ST_AbstractBinaryDrive_Status :
STRUCT
	Running   : BOOL;
	Active    : BOOL;
	Forward   : BOOL;
	Backward  : BOOL;
	Error     : BOOL;
	ErrorCode : UDINT;
END_STRUCT
END_TYPE

// ---- Library/DUTs/ST_AbstractBinaryDrive_HMI.TcDUT
// Conveyor drive HMI interface - ONE struct per tile.
// Extends ST_ComponentBase_HMI, so one bound parameter also carries Config,
// Command and Status - and the added members may not reuse those three names.
//
// The one unit type here with a real device command block: a drive has no SPT
// component of its own, so DeviceCommand is it. Used by Transport01, Transport02
// and both lift carriage belts.
TYPE ST_AbstractBinaryDrive_HMI EXTENDS ST_ComponentBase_HMI :
STRUCT
	DeviceConfig	: ST_AbstractBinaryDrive_Config;
	DeviceCommand	: ST_AbstractBinaryDrive_Command;
	Device			: ST_AbstractBinaryDrive_Status;
END_STRUCT
END_TYPE

// ---- Library/DUTs/ST_BaseModule_HMI.TcDUT
// The one HMI interface every module in this project publishes.
// Extends the SPT module struct, so a tile gets Config, Command and Status in the
// shape the framework already maintains.
//
// The base FB owns its own PackMLBaseModule_HMI and fills it; this is the
// PUBLISHED MIRROR. The module bridges them in HMICommunication (commands, before
// state control) and PublishHMI (status, after). NEITHER HALF IS OPTIONAL: without
// the command push the panel's buttons reach nothing, without the status pull the
// tile reads zeros.
//
// A descendant adds exactly one member, and it must NOT be named Config, Command,
// Status or Sequence - redeclaring an inherited member is a compile error.
TYPE ST_BaseModule_HMI EXTENDS ST_PackMLBaseModule_HMI :
STRUCT
	Sequence : ST_Sequence_Status;
	// The PackML state as text. ST_PackMLBaseModule_Status carries State as an
	// enum only, and tchmiconfig.json sets binding.symbolError to "Ignore", so a
	// client side enum conversion that fails to resolve renders an empty control
	// and reports nothing. See F_PMLStateName.
	StateName : STRING(20);
END_STRUCT
END_TYPE

// ---- Library/DUTs/ST_Sequence_Status.TcDUT
TYPE ST_Sequence_Status :
STRUCT
	StepIndex 			: UDINT;
	StepName 			: STRING(20);
END_STRUCT
END_TYPE

// ---- Library/DUTs/ST_FG_System_Safety.TcDUT
// The safety chain, broken out for the panel.
// GuardsSecure and EmergencyStopActive are the two facts the machine consumes;
// the rest exists so an operator can see WHICH door or mushroom is holding the
// cell, which the composed booleans cannot say.
// Door array order is fixed and matches the twin:
//   [1] B_SafetyDoor11  [2] B_SafetyDoor12  [3] B_SafetyDoor13   (side 1)
//   [4] B_SafetyDoor21  [5] B_SafetyDoor22  [6] B_SafetyDoor23   (side 2)
TYPE ST_FG_System_Safety :
STRUCT
	// The composed chain. Guards are only enforced in Production; the machine
	// applies that rule, not this struct.
	GuardsSecure : BOOL;
	EmergencyStopActive : BOOL;

	// TRUE while the PLC is commanding every lock engaged, i.e. in Production.
	DoorsRequestedLocked : BOOL;

	DoorClosed : ARRAY[1..6] OF BOOL;
	DoorLocked : ARRAY[1..6] OF BOOL;
	// 0 none, 1 lock commanded but never confirmed.
	DoorFaultCode : ARRAY[1..6] OF UDINT;

	EStopActive : ARRAY[1..2] OF BOOL;
END_STRUCT
END_TYPE

// ---- Library/DUTs/ST_IlluminatedButton_Config.TcDUT
TYPE ST_IlluminatedButton_Config :
STRUCT
	// Contact polarity. TRUE means the input is NORMALLY CLOSED - it reads TRUE
	// while healthy and FALSE while pressed - which is how a real emergency stop
	// is wired, and how SIM_1 presents the twin's buttons. Both mushrooms set it
	// TRUE. Surfaced on the panel because getting it wrong is invisible and
	// dangerous - see _workflow/reference/plc-io-exceptions.md.
	Inverted : BOOL;
END_STRUCT
END_TYPE

// ---- Library/DUTs/ST_IlluminatedButton_Status.TcDUT
TYPE ST_IlluminatedButton_Status :
STRUCT
	// TRUE while pressed. On the emergency stops this means LATCHED - the twin's
	// mushrooms are Toggle type, so a click holds until clicked again.
	Active	: BOOL;
	// The lamp as the PLC is driving it this scan. Solid while latched, flashing
	// while latched during Clearing - the owning module decides, not this device.
	Lamp	: BOOL;
END_STRUCT
END_TYPE

// ---- Library/DUTs/ST_IlluminatedButton_HMI.TcDUT
// Illuminated button HMI interface - ONE struct per tile.
// Extends ST_ComponentBase_HMI, so one bound parameter also carries Config,
// Command and Status - and the added members may not reuse those three names.
//
// NO DeviceCommand: the lamp is driven by the owning module from the machine's
// PackML state, and a panel able to override it could make a latched emergency
// stop look released.
TYPE ST_IlluminatedButton_HMI EXTENDS ST_ComponentBase_HMI :
STRUCT
	DeviceConfig	: ST_IlluminatedButton_Config;
	Device			: ST_IlluminatedButton_Status;
END_STRUCT
END_TYPE

// ---- Library/DUTs/ST_SafetyDoor_Config.TcDUT
TYPE ST_SafetyDoor_Config :
STRUCT
	// How long the lock has to confirm after being commanded before fault 1 is
	// raised. Writable from the panel: a sticky lock on a demo cell is exactly the
	// kind of thing tuned against the running machine.
	LockTime : TIME;
END_STRUCT
END_TYPE

// ---- Library/DUTs/ST_SafetyDoor_Status.TcDUT
TYPE ST_SafetyDoor_Status :
STRUCT
	// The two bits that matter, and they are NOT redundant: a door can be shut
	// without being locked, and that is precisely the state that must not let
	// Production start.
	Closed	: BOOL;
	Locked	: BOOL;

	// Closed AND Locked. Published as its own bit so a panel shows the same
	// verdict the safety chain uses instead of ANDing two lamps by eye.
	Secure	: BOOL;

	// TRUE while the PLC is commanding this lock engaged - Production only.
	LockRequested : BOOL;

	// 0 none, 1 lock commanded but never confirmed within LockTime.
	FaultCode : UDINT;
END_STRUCT
END_TYPE

// ---- Library/DUTs/ST_SafetyDoor_HMI.TcDUT
// Safety door HMI interface - ONE struct per tile.
// Extends ST_ComponentBase_HMI, so one bound parameter also carries Config,
// Command and Status - and the added members may not reuse those three names.
//
// NO DeviceCommand, deliberately. The lock is commanded by FG_System from the
// machine's PackML mode, and a panel able to override that could unlock a running
// cell. FG_System.HMI.Safety carries the same facts as arrays for a whole-cell
// summary; this struct is for a per-door tile.
TYPE ST_SafetyDoor_HMI EXTENDS ST_ComponentBase_HMI :
STRUCT
	DeviceConfig	: ST_SafetyDoor_Config;
	Device			: ST_SafetyDoor_Status;
END_STRUCT
END_TYPE

// ---- Library/DUTs/ST_SignalTower_Config.TcDUT
TYPE ST_SignalTower_Config :
STRUCT
	// Half period of the flash clock. Writable from the panel, which is the only
	// practical way to tune a blink rate against a running machine.
	FlashTime : TIME;
END_STRUCT
END_TYPE

// ---- Library/DUTs/ST_SignalTower_Status.TcDUT
TYPE ST_SignalTower_Status :
STRUCT
	// The four lamps exactly as the coils are being driven this scan - already
	// blended, so a flashing lamp reads TRUE/FALSE at the flash rate and a panel
	// bound to these mirrors the real tower without re-deriving anything.
	Red		: BOOL;
	Yellow	: BOOL;
	Blue	: BOOL;
	Green	: BOOL;

	// The shared flash phase, for a panel that wants to blink something in step
	// with the tower rather than run its own clock.
	Flash	: BOOL;

	// The conditions behind the lamps, so a panel can say WHY a lamp is lit
	// instead of leaving the operator to infer it from a colour. Amber and blue
	// have no source in this machine yet and stay FALSE - see
	// _workflow/reference/state-lamp.md.
	StarvedUpstream		: BOOL;
	BlockedDownstream	: BOOL;
	LowMaterial			: BOOL;
	MaterialExhausted	: BOOL;
END_STRUCT
END_TYPE

// ---- Library/DUTs/ST_SignalTower_HMI.TcDUT
// Signal tower HMI interface - ONE struct per tile.
// Extends ST_ComponentBase_HMI, so one bound parameter also carries Config,
// Command and Status - and the added members may not reuse those three names.
//
// NO DeviceCommand: the lamps derive from the machine's PackML state and nothing
// else may drive them.
TYPE ST_SignalTower_HMI EXTENDS ST_ComponentBase_HMI :
STRUCT
	DeviceConfig	: ST_SignalTower_Config;
	Device			: ST_SignalTower_Status;
END_STRUCT
END_TYPE

// ---- Library/DUTs/ST_HMI_FG_System.TcDUT
// FG_System's HMI contract.
//
// ST_BaseModule_HMI's header states the constraint: a descendant adds exactly one
// member, and it must not be named Config, Command, Status or Sequence, because
// redeclaring an inherited member is a compile error. That member is Safety.
TYPE ST_HMI_FG_System EXTENDS ST_BaseModule_HMI :
STRUCT
	Safety : ST_FG_System_Safety;
END_STRUCT
END_TYPE

// ---- Library/DUTs/ST_AbstractCamera_Command.TcDUT
// What an operator may ask of a camera from the panel, in Manual and Maintenance.
// One member per control bit, so the panel never has to know the bit layout.
//
// Two signals, not three. The light was folded away when the device moved to a
// real vision-sensor interface: a camera of this kind switches its own
// illumination with the shot, and a separate lamp bit was modelling a lamp this
// device does not have.
TYPE ST_AbstractCamera_Command :
STRUCT
	Enable	: BOOL;
	Trigger	: BOOL;
END_STRUCT
END_TYPE

// ---- Library/DUTs/ST_AbstractCamera_Status.TcDUT
// What the camera reports back - four real signals off the status byte, none of
// them inferred from the control side. Ready is permission to trigger, Busy is the
// shot in progress, ResultValid says a verdict is on the wire now.
//
// READ ResultOK ONLY WHILE ResultValid. Outside that window it is FALSE because
// there is no verdict, not because the part was bad.
TYPE ST_AbstractCamera_Status :
STRUCT
	Ready		: BOOL;
	Busy		: BOOL;
	ResultValid	: BOOL;
	ResultOK	: BOOL;
END_STRUCT
END_TYPE

// ---- Library/DUTs/ST_AbstractCamera_HMI.TcDUT
// Camera HMI interface - ONE struct per tile.
//
// Extends ST_ComponentBase_HMI, so Config, Command and Status arrive inherited
// and the added members cannot reuse those three names. Same shape as
// ST_AbstractLightSource_HMI, which is the component this one was modelled on.
TYPE ST_AbstractCamera_HMI EXTENDS ST_ComponentBase_HMI :
STRUCT
	DeviceCommand	: ST_AbstractCamera_Command;
	Device			: ST_AbstractCamera_Status;
END_STRUCT
END_TYPE

// ---- Library/DUTs/ST_AbstractBunker_Command.TcDUT
// The two control bits, one member each, so the panel never handles a bit index.
// They are separate because the vibration table and the feed conveyor are
// separate machines - running the table into a stopped conveyor is a way to jam
// the pick position, and a commissioning engineer needs to be able to do one
// without the other.
TYPE ST_AbstractBunker_Command :
STRUCT
	RunTable	: BOOL;
	RunConveyor	: BOOL;
END_STRUCT
END_TYPE

// ---- Library/DUTs/ST_AbstractBunker_Status.TcDUT
// THE BUNKER REPORTS NOTHING BACK. Its status byte is unused in the twin, so
// every field here is the commanded state read off the control byte, not a
// measurement. A tile bound to this shows what the PLC is asking for; it cannot
// show whether the table is actually turning, because nothing on this device
// says so.
TYPE ST_AbstractBunker_Status :
STRUCT
	TableRunning	: BOOL;
	ConveyorRunning	: BOOL;
END_STRUCT
END_TYPE

// ---- Library/DUTs/ST_AbstractBunker_HMI.TcDUT
// Bunker HMI interface - ONE struct per tile.
//
// Extends ST_ComponentBase_HMI, so Config, Command and Status arrive inherited
// and the added members cannot reuse those three names.
TYPE ST_AbstractBunker_HMI EXTENDS ST_ComponentBase_HMI :
STRUCT
	DeviceCommand	: ST_AbstractBunker_Command;
	Device			: ST_AbstractBunker_Status;
END_STRUCT
END_TYPE

// ---- Modules/11 FG_01/ST_FG_01_Identify_Status.TcDUT
// What the identification has to say beyond the PackML state.
//
// THE SAME THREE FAULT CODES AS ST_FG_02_Inspection_Status, deliberately - both
// stations now drive the same device through the same handshake, and an operator
// should not have to learn two numbering schemes for one failure:
//
//   1  NOK       - the camera returned a serial number and it was not the one
//                  this station expects
//   2  not ready - Enable was set and Ready never came: the camera is not
//                  answering at all, which is a wiring or device fault
//   3  no result - the shot was triggered and no verdict arrived in time: the
//                  camera is there but the exposure never completed
//
// FG_01 HAD NO FAULT CODE AT ALL until the reader became a camera. It could not
// have had one: the old reader's status bit was an echo of the trigger,
// the sequence held the window open for a fixed 1 s and moved on whatever came
// back, and there was nothing to report. A real verdict that nobody consumes is
// worse than no verdict, so this is what consumes it.
//
// LastResultOK is the verdict from the most recent completed read, latched so the
// panel still shows it after ResultValid has dropped. It is not a fault - a NOK
// sets code 1 as well.
//
// Cleared in FG_01.Clearing.
TYPE ST_FG_01_Identify_Status :
STRUCT
	FaultCode		: DINT;
	LastResultOK	: BOOL;
END_STRUCT
END_TYPE

// ---- Modules/11 FG_01/ST_HMI_FG_01.TcDUT
// FG_01 HMI interface - ONE struct for the group tile.
//
// Extends ST_BaseModule_HMI, so it inherits the whole SPT module interface:
//   Config.Name / LogStateChanges / LogModeChanges / ModeNames
//   Command.Mode / State / Activate*Log / Deactivat*Log      (writable)
//   Status.Busy / Error / ErrorID / Mode / State / HMIControlAvailable
//   Sequence.StepIndex / StepName
//   StateName
//
// The one added member CANNOT be called Config, Command, Status or Sequence -
// those are inherited and redeclaring them is a compile error. Hence Identify.
//
// FG_01 bound a plain ST_BaseModule_HMI while its reader had a status bit that
// echoed the trigger: there was no group-level fact that no device already owned.
// A real verdict and three distinguishable failure modes are exactly such a fact.
// Same shape as ST_HMI_FG_02, which is the struct this one was modelled on.
TYPE ST_HMI_FG_01 EXTENDS ST_BaseModule_HMI :
STRUCT
	Identify	: ST_FG_01_Identify_Status;
END_STRUCT
END_TYPE

// ---- Modules/12 FG_02/ST_FG_02_Inspection_Status.TcDUT
// What the inspection has to say beyond the PackML state.
//
// THREE FAULT CODES, one per way the handshake can fail, and no more. Each is a
// distinct thing an operator would do something different about:
//
//   1  NOK      - the camera returned a verdict and it was bad
//   2  not ready - Enable was set and Ready never came: the camera is not
//                  answering at all, which is a wiring or device fault
//   3  no result - the shot was triggered and no verdict arrived in time: the
//                  camera is there but the exposure never completed
//
// Telling 2 from 3 is the whole reason the interface grew from one status bit to
// four. The old device could only ever say nothing.
//
// LastResultOK is the verdict from the most recent completed shot, latched so the
// panel still shows it after ResultValid has dropped. It is not a fault - a NOK
// sets code 1 as well.
//
// Cleared in FG_02.Clearing.
TYPE ST_FG_02_Inspection_Status :
STRUCT
	FaultCode		: DINT;
	LastResultOK	: BOOL;
END_STRUCT
END_TYPE

// ---- Modules/12 FG_02/ST_HMI_FG_02.TcDUT
// FG_02 HMI interface - ONE struct for the group tile.
//
// Extends ST_BaseModule_HMI, so it inherits the whole SPT module interface:
//   Config.Name / LogStateChanges / LogModeChanges / ModeNames
//   Command.Mode / State / Activate*Log / Deactivat*Log      (writable)
//   Status.Busy / Error / ErrorID / Mode / State / HMIControlAvailable
//   Sequence.StepIndex / StepName
//   StateName
//
// The one added member CANNOT be called Config, Command, Status or Sequence -
// those are inherited and redeclaring them is a compile error. Hence Inspection.
//
// FG_02 did not need this while its camera had a single status bit that echoed the
// trigger: there was no group-level fact that no device already owned. A real
// verdict and three distinguishable failure modes are exactly such a fact.
TYPE ST_HMI_FG_02 EXTENDS ST_BaseModule_HMI :
STRUCT
	Inspection	: ST_FG_02_Inspection_Status;
END_STRUCT
END_TYPE

// ---- Modules/13 FG_03/ST_FG_03_Transfer_Status.TcDUT
// What the two grip sensors have to say beyond the PackML state.
//
// FG_03 HAD NO FAULT CODE AT ALL until B_Detect1 and B_Detect2 arrived, because it
// had nothing to report: every step waited on a cylinder limit, and a cylinder
// limit cannot fail in a way the cylinder itself does not already alarm. A part
// sensor can - it is the first thing in this group that can disagree with the
// actuators.
//
//   1  stuck at   - Resetting could not separate the two grippers in the handover
//      handover     window: arm 2 reported its jaws open and B_Detect2 still saw
//                   the part. Nothing was moved, because every way out of that
//                   window pulls the two arms apart with one part between them.
//                   The arms are still standing at the handover; free the part by
//                   hand, then Clear and Reset.
//   2  no pick    - Y_Gripper2 closed on slot 1 and B_Detect2 never confirmed a
//                   part. An empty slot, a mispositioned pallet, or a grip that
//                   closed on nothing - which reaches its extended limit SOONER
//                   than a real grip, so the limit alone cannot tell them apart.
//   3  no handover- Y_Gripper1 closed at the handover and B_Detect1 never confirmed.
//                   This is the dangerous one: without it, step 90 opens arm 2
//                   against a grip that was never made and the part falls.
//   4  no release - a gripper opened and its sensor still sees the part, inside
//                   Execute. The part is jammed in the jaws.
//   5  off safe   - a cycle was started with a part held by an arm that is NOT at
//                   its safe position (X and Y retracted). The resume entry point
//                   is derived from which gripper is full, and it is only right if
//                   the arm is where the reset would have parked it. Someone jogged
//                   it in Manual, or code 1 is standing. Reset fixes it, because
//                   Resetting reaches a safe position from anywhere.
//
// WHY CODE 1 DOES NOT ABORT OUT OF Resetting. A reset must terminate on time and on
// its own cylinders - transport-behaviour.md 4, learned twice the expensive way.
// Aborting mid-reset would leave the arms wherever they happened to be, which is
// worse than stopping cleanly and saying so. Resetting completes; Execute refuses
// the next cycle through code 5, because a part stuck at the handover is by
// definition not at a safe position.
//
// ResumePoint is not a fault. It is which sub-sequence the NEXT Start will enter,
// derived every scan from the two grip sensors - the same derivation Execute step 0
// makes, published so the panel can show it before anyone presses anything:
//
//   1  the whole cycle, from the pick out of slot 1  (both grippers empty)
//   2  the handover, from arm 2's safe position      (B_Detect2)
//   3  the placement into slot 2, from arm 1's       (B_Detect1)
//
// Cleared in FG_03.Clearing - the fault code, that is. ResumePoint is derived and
// has nothing to clear.
TYPE ST_FG_03_Transfer_Status :
STRUCT
	FaultCode	: DINT;
	ResumePoint	: DINT;
END_STRUCT
END_TYPE

// ---- Modules/13 FG_03/ST_HMI_FG_03.TcDUT
// FG_03 HMI interface - ONE struct for the group tile.
//
// Extends ST_BaseModule_HMI, so it inherits the whole SPT module interface:
//   Config.Name / LogStateChanges / LogModeChanges / ModeNames
//   Command.Mode / State / Activate*Log / Deactivat*Log      (writable)
//   Status.Busy / Error / ErrorID / Mode / State / HMIControlAvailable
//   Sequence.StepIndex / StepName
//   StateName
//
// The one added member CANNOT be called Config, Command, Status or Sequence -
// those are inherited and redeclaring them is a compile error. Hence Transfer.
//
// FG_03 used the bare ST_BaseModule_HMI until it acquired something of its own to
// say. Same shape as ST_HMI_FG_01, ST_HMI_FG_02, ST_HMI_FG_04 and ST_HMI_FG_05.
TYPE ST_HMI_FG_03 EXTENDS ST_BaseModule_HMI :
STRUCT
	Transfer	: ST_FG_03_Transfer_Status;
END_STRUCT
END_TYPE

// ---- Modules/14 FG_04/ST_FG_04_Press_Status.TcDUT
// What the press has to say beyond the PackML state.
//
// ONE FAULT CODE, not a set of six like the transport stations. FG_04 has exactly
// one condition worth reporting - the press bottomed out with nothing correctly
// seated - and padding the enumeration out to look like FB_TransferIndex's would
// be inventing failure modes this station does not have.
//
//   1  NIO - press reached its bottom limit and B_NIO reports no part seated
//
// Cleared in FG_04.Clearing, alongside the component resets.
TYPE ST_FG_04_Press_Status :
STRUCT
	FaultCode	: DINT;
END_STRUCT
END_TYPE

// ---- Modules/14 FG_04/ST_HMI_FG_04.TcDUT
// FG_04 HMI interface - ONE struct for the group tile.
//
// Extends ST_BaseModule_HMI, so it inherits the whole SPT module interface:
//   Config.Name / LogStateChanges / LogModeChanges / ModeNames
//   Command.Mode / State / Activate*Log / Deactivat*Log      (writable)
//   Status.Busy / Error / ErrorID / Mode / State / HMIControlAvailable
//   Sequence.StepIndex / StepName
//   StateName
//
// The one added member CANNOT be called Config, Command, Status or Sequence -
// those are inherited and redeclaring them is a compile error. Hence Press.
//
// FG_04 is the only one of the five station groups that needs an extension at
// all. The other four publish ST_BaseModule_HMI unchanged, because every device
// they own publishes itself and there is no group-level fact left over. Here
// there is one: B_NIO's verdict outlives the sensor reading that produced it.
TYPE ST_HMI_FG_04 EXTENDS ST_BaseModule_HMI :
STRUCT
	Press	: ST_FG_04_Press_Status;
END_STRUCT
END_TYPE

// ---- Modules/15 FG_05/ST_FG_05_Capping_Status.TcDUT
// What the identification read has to say beyond the PackML state.
//
// THE READ IS OF THE ASSEMBLY, NOT THE CAP. The camera returns the assembly's
// CapsID - which cap that assembly wants - and the station fits one only to an
// assembly of the type it is set up for.
//
// THE SAME THREE FAULT CODES AS FG_01 AND FG_02, deliberately. All three stations
// drive the same FB_AbstractCamera through the same handshake, and an operator
// should not have to learn three numbering schemes for one device:
//
//   1  NOK       - the camera returned a CapsID and it was not the one this
//                  station caps: the wrong assembly, or an empty pallet
//   2  not ready - Enable was set and Ready never came: the camera is not
//                  answering at all, which is a wiring or device fault
//   3  no result - the shot was triggered and no verdict arrived in time: the
//                  camera is there but the exposure never completed
//
// CODES 4 TO 6 ARE THE GRIPPER'S, not the camera's, and they arrived with B_Detect,
// the grip sensor. They share this struct rather than getting their own because an
// operator reads one number off one tile:
//
//   4  off safe   - a cycle was started with a cap held by a unit that is NOT at the
//                   safe position (X max, both Z min). The resume entry point is
//                   derived from the fact that a cap is held, and it is only right
//                   if the unit is where the reset would have parked it. Someone
//                   jogged an axis in Manual. Reset fixes it, because Resetting
//                   reaches the safe position from anywhere.
//
//                   A cap held AT the safe position is not a fault at all - it is a
//                   resumable cycle, and Resetting raises nothing for it.
//   5  no pick    - the jaws closed at the pick position and no cap appeared in
//                   them. B_Part said a cap was THERE; B_Detect says none is HELD.
//                   A crooked cap, or one that moved as the jaws closed.
//   6  no release - the jaws opened over the part and the cap is still in them.
//                   Lifting now would carry it back off the pallet and send an
//                   uncapped assembly on with nothing having complained.
//
// FG_05 HAD NO FAULT CODE AT ALL while its reader's status bit was an echo of the
// trigger. Step 20 took the read, left on it OR a 1 s timeout, and branched on
// neither - there was nothing to report.
//
// THE ABORT COSTS MORE HERE THAN IT DOES IN FG_01 OR FG_02, and that is why the
// read sits where it does. It runs BEFORE the gripper has taken anything, so an
// abort leaves the cap in the feed and the handling unit empty and home. Moving
// the read later would abort with a cap held in the air over the pallet.
//
// LastResultOK is the verdict from the most recent completed read, latched so the
// panel still shows it after ResultValid has dropped. It is not a fault - a NOK
// sets code 1 as well.
//
// ResumePoint is not a fault. It is which part of the cycle the NEXT Start will
// enter, derived every scan from B_Detect - the same derivation Execute step 0
// makes, published so the panel can show it before anyone presses anything:
//
//   1  the whole cycle, from the camera read and the pick   (jaws empty)
//   2  the placement, from the safe position over the pallet (cap held)
//
// FG_03 publishes the same field with three values; this station has one gripper
// and therefore one place to resume from.
//
// Cleared in FG_05.Clearing - the fault code, that is. ResumePoint is derived and
// has nothing to clear.
TYPE ST_FG_05_Capping_Status :
STRUCT
	FaultCode		: DINT;
	ResumePoint		: DINT;
	LastResultOK	: BOOL;
END_STRUCT
END_TYPE

// ---- Modules/15 FG_05/ST_HMI_FG_05.TcDUT
// FG_05 HMI interface - ONE struct for the group tile.
//
// Extends ST_BaseModule_HMI, so it inherits the whole SPT module interface:
//   Config.Name / LogStateChanges / LogModeChanges / ModeNames
//   Command.Mode / State / Activate*Log / Deactivat*Log      (writable)
//   Status.Busy / Error / ErrorID / Mode / State / HMIControlAvailable
//   Sequence.StepIndex / StepName
//   StateName
//
// The one added member CANNOT be called Config, Command, Status or Sequence -
// those are inherited and redeclaring them is a compile error. Hence Capping.
//
// Same shape as ST_HMI_FG_01 and ST_HMI_FG_02. The three camera stations now
// publish the same two facts under three names that say which station it is -
// Identify, Inspection, Capping - rather than one shared name that would say
// nothing on any of them.
TYPE ST_HMI_FG_05 EXTENDS ST_BaseModule_HMI :
STRUCT
	Capping	: ST_FG_05_Capping_Status;
END_STRUCT
END_TYPE

// ---- Modules/10 FG_Transport/ST_TransferIndex_HMI.TcDUT
// Index unit HMI interface - ONE struct per tile.
//
// Extends ST_BaseModule_HMI, so it inherits the whole SPT module interface:
//   Config.Name / LogStateChanges / LogModeChanges / ModeNames
//   Command.Mode / State / Activate*Log / Deactivat*Log      (writable)
//   Status.Busy / Error / ErrorID / Mode / State / HMIControlAvailable
//   Sequence.StepIndex / StepName
//   StateName
// FB_TransferIndex.HMICommunication bridges Command into the base's own
// PackMLBaseModule_HMI before the base acts on it, and PublishHMI copies Config
// and Status back out afterwards.
//
// The one added member CANNOT be called Config, Command, Status or Sequence -
// those are inherited and redeclaring them is a compile error. Hence Station.
//
// There is still no per-device command block here: an index unit is jogged
// through its two SPT components, which own their command structs themselves -
//   MAIN.Machine.FG_Transport.Index03.Y_Stopper.SolenoidHMI.Command.Extend
//   MAIN.Machine.FG_Transport.Index03.Y_Lift.SolenoidHMI.Command.Extend
TYPE ST_TransferIndex_HMI EXTENDS ST_BaseModule_HMI :
STRUCT
	Station	: ST_TransferIndex_Status;
END_STRUCT
END_TYPE

// ---- Modules/10 FG_Transport/ST_TransferIndex_Status.TcDUT
// What an index unit publishes BEYOND what the SPT base already gives it.
//
// State, StateName, SequenceState and HMIControlAvailable used to live here and
// have all been removed: ST_TransferIndex_HMI extends ST_BaseModule_HMI, so they
// arrive inherited from ST_PackMLBaseModule_Status and ST_BaseModule_HMI.
// Duplicating them meant two copies of the same truth kept in step by hand.
//
// Everything left is genuinely this unit type's own.
TYPE ST_TransferIndex_Status :
STRUCT
	// --- Ring handshake -----------------------------------------------------
	// Ready: idle and empty, will accept a pallet.
	// Occupied: holding a pallet. Deliberately not called Busy - the base FB
	// already uses Busy to mean "mid async operation", which is something else.
	Ready				: BOOL;
	Occupied			: BOOL;
	NextReady			: BOOL;
	SendToNext			: BOOL;

	// --- Functional group handshake -----------------------------------------
	// ReadyForOperation: pallet stopped AND lifted, the group may run.
	// OperationDone: the group has reported finished.
	ReadyForOperation	: BOOL;
	OperationDone		: BOOL;

	// --- Diagnostics --------------------------------------------------------
	// 0 none  1 no home  2 lift did not raise  3 group did not finish
	// 4 lift did not lower  5 no release  6 pallet never reached the exit sensor
	FaultCode			: DINT;
END_STRUCT
END_TYPE

// ---- Modules/10 FG_Transport/ST_TransferLift_HMI.TcDUT
// Lift unit HMI interface - ONE struct per tile.
//
// Extends ST_BaseModule_HMI, so Config, Command, Status, Sequence and StateName
// all arrive inherited from the SPT module interface. See ST_TransferIndex_HMI
// for the full member list and the bridge that keeps it current.
//
// The carriage belt publishes itself: M_Conveyor is an FB_AbstractBinaryDrive and
// carries its own ST_AbstractBinaryDrive_HMI at
//   MAIN.Machine.FG_Transport.Lift01.M_Conveyor.HMI
// which the tile binds as a second parameter. The two cylinders are jogged
// through their own SolenoidHMI structs.
TYPE ST_TransferLift_HMI EXTENDS ST_BaseModule_HMI :
STRUCT
	Station	: ST_TransferLift_Status;
END_STRUCT
END_TYPE

// ---- Modules/10 FG_Transport/ST_TransferLift_Status.TcDUT
// What a lift unit publishes BEYOND what the SPT base already gives it.
// State, StateName, SequenceState and HMIControlAvailable are inherited through
// ST_TransferLift_HMI EXTENDS ST_BaseModule_HMI and are no longer duplicated.
TYPE ST_TransferLift_Status :
STRUCT
	// --- Ring handshake -----------------------------------------------------
	// A lift is a pulling station: it has no SendToNext. PayloadIncoming is how
	// the predecessor announces a pallet.
	Ready				: BOOL;
	Occupied			: BOOL;
	NextReady			: BOOL;
	PayloadIncoming		: BOOL;

	// FALSE = this lift raises (Lift01), TRUE = it lowers (Lift02). Published so
	// a tile can label its travel buttons without knowing which instance it is.
	ReverseDirection	: BOOL;

	// --- Diagnostics --------------------------------------------------------
	// 0 none  1 no home  2 pallet never arrived aboard  3 travel failed
	// 4 pallet never left
	FaultCode			: DINT;
END_STRUCT
END_TYPE

// ---- Modules/10 FG_Transport/ST_TransferStopper_HMI.TcDUT
// Stopper unit HMI interface - ONE struct per tile.
//
// Extends ST_BaseModule_HMI, so Config, Command, Status, Sequence and StateName
// all arrive inherited from the SPT module interface. See ST_TransferIndex_HMI
// for the full member list and the bridge that keeps it current.
//
// Still no command block of its own: a stopper is jogged through its one SPT
// component - MAIN.Machine.FG_Transport.Stopper02.Y_Stopper.SolenoidHMI.Command.Extend
TYPE ST_TransferStopper_HMI EXTENDS ST_BaseModule_HMI :
STRUCT
	Station	: ST_TransferStopper_Status;
END_STRUCT
END_TYPE

// ---- Modules/10 FG_Transport/ST_TransferStopper_Status.TcDUT
// What a stopper unit publishes BEYOND what the SPT base already gives it.
// State, StateName, SequenceState and HMIControlAvailable are inherited through
// ST_TransferStopper_HMI EXTENDS ST_BaseModule_HMI and are no longer duplicated.
TYPE ST_TransferStopper_Status :
STRUCT
	// --- Ring handshake -----------------------------------------------------
	Ready				: BOOL;
	Occupied			: BOOL;
	NextReady			: BOOL;
	SendToNext			: BOOL;

	// --- Diagnostics --------------------------------------------------------
	// 0 none  1 no block  2 no release  3 pallet never reached the exit sensor
	FaultCode			: DINT;
END_STRUCT
END_TYPE

// ---- POUs/MAIN.TcPOU
PROGRAM MAIN
VAR
	Machine			: Machine := (Name := 'OC Demo 1', LogStateChanges := TRUE);

	//Local TwinCAT HMI
	{ attribute 'TcHmiSymbol.AddSymbol' }
	ControlSource_HMI_Web	: FB_ControlSource_HMI;

	// The physical operator panel, H_ControlPanel. A second control source rather
	// than a device: FB_ControlSource already owns the START/STOP/RESET ladder,
	// and MAX_NO_OF_EXTERNAL_CONTROLLERS is an array, so the two coexist.
	{ attribute 'TcHmiSymbol.AddSymbol' }
	ControlSource_Panel		: FB_ControlSource_Panel;

	InitComplete	: BOOL;
END_VAR

CyclicLogic();

METHOD CyclicLogic
VAR_INPUT
END_VAR
IF NOT InitComplete THEN
	InitComplete := Initialize();
	RETURN;
END_IF

// The panel's two inputs from the machine, before it runs on them. SafetyOk
// vetoes its Start and Reset permissives, so a button whose press would be
// refused stays dark instead of inviting it; Flash is the signal tower's clock,
// shared so every flashing lamp on the machine blinks in phase.
ControlSource_Panel.SafetyOk	:= Machine.SafetyOk;
ControlSource_Panel.Flash		:= Machine.IndicationFlash;

// Control sources first, so this scan's requests become PackML commands before
// the state machine runs on them.
ControlSource_HMI_Web.CyclicLogic();
ControlSource_Panel.CyclicLogic();

Machine.CyclicLogic();
END_METHOD

METHOD Initialize : BOOL
VAR_INPUT
END_VAR
// Top level machine initialization. Every deeper layer of modules is named inside
// its own parent's Initialize; only the machine itself is named here.
_AppInfo.KeepOutputsOnBP := TRUE;

// Registration hands the control source an interface to the machine, which is
// what its inherited Registered property reports on.
IF NOT ControlSource_HMI_Web.Registered THEN
	Machine.RegisterExternalController(ControlSource_HMI_Web);
END_IF

IF NOT ControlSource_Panel.Registered THEN
	Machine.RegisterExternalController(ControlSource_Panel);
END_IF

ControlSource_HMI_Web.CyclicLogic();
ControlSource_Panel.CyclicLogic();

Initialize := TRUE;
END_METHOD

END_PROGRAM

// ---- Modules/00 Machine/Machine.TcPOU
// Machine - the top level module. Owns the PackML mode and the safety policy,
// and brokers the Index <-> functional group handshakes every scan.
// EnforceSafety aborts on NOT SafetyOk, EXCEPT in Aborting/Aborted/Clearing -
// re-issuing the abort there is a deadlock the machine cannot leave.
// Contract: _workflow/reference/fg-system-safety.md
FUNCTION_BLOCK Machine EXTENDS FB_PackML_BaseModule
VAR
	FG_System : FG_System := (Name := 'FG_System', LogStateChanges := TRUE);
	FG_Transport : FG_Transport := (Name := 'FG_Transport', LogStateChanges := TRUE);

	// The five processing groups, in ring order. Each one is served by the index
	// unit of the same number and by no other - see BrokerIndexHandshakes.
	FG_01 : FG_01 := (Name := 'FG_01', LogStateChanges := TRUE);
	FG_02 : FG_02 := (Name := 'FG_02', LogStateChanges := TRUE);
	FG_03 : FG_03 := (Name := 'FG_03', LogStateChanges := TRUE);
	FG_04 : FG_04 := (Name := 'FG_04', LogStateChanges := TRUE);
	FG_05 : FG_05 := (Name := 'FG_05', LogStateChanges := TRUE);
END_VAR

ACTION BrokerIndexHandshakes:
// Index unit -> functional group, brokered.
// The index units and the groups are sibling submodules, so this is where the
// two halves meet - neither reaches into the other.
//   1. the index reports ReadyForOperation once the pallet is stopped AND lifted
//   2. the group runs its operation
//   3. the group reports complete, and the index clears the flag itself
// A group that is not running is answered IMMEDIATELY, so the ring keeps turning
// whichever group is missing. There is no bypass flag and none is needed.

BrokerGroup(Index := 1, Group := FG_01);
BrokerGroup(Index := 2, Group := FG_02);
BrokerGroup(Index := 3, Group := FG_03);
BrokerGroup(Index := 4, Group := FG_04);
BrokerGroup(Index := 5, Group := FG_05);
END_ACTION

// One index unit, one functional group, one handshake. Called once per group from
// BrokerIndexHandshakes, every scan.
// The five groups share no base but FB_PackML_BaseModule, so the only thing that
// can hold all of them is I_PackML_BaseModule.
// LIVENESS IS READ OFF THE STATE, NOT OFF InitComplete. An unregistered module
// never has CyclicLogic() called, so it never leaves ePMLState_Undefined - a
// direct test of whether its state machine is running. InitComplete was a proxy,
// and is not on the interface.
METHOD PRIVATE BrokerGroup
VAR_INPUT
	Index	: INT;						// 1..5, the index unit that serves this group
	Group	: I_PackML_BaseModule;		// the group it serves
END_VAR
IF NOT FG_Transport.IsIndexReadyForOperation(Index) THEN
	RETURN;
END_IF

// Not there, or not running. Answer for it so the pallet is released rather than
// held until the index unit's operation timeout raises fault 3.
IF Group = 0 OR_ELSE Group.CurrentState = E_PMLState.ePMLState_Undefined THEN
	FG_Transport.SetIndexOperationDone(Index := Index, Value := TRUE);
	RETURN;
END_IF

CASE Group.CurrentState OF

	E_PMLState.ePMLState_Idle:
		// Pallet stopped and lifted. Run.
		Group.ChangeState(E_PMLCommand.ePMLCommand_Start);

	E_PMLState.ePMLState_Complete:
		// Finished. Release the pallet and put the group back to Idle for the
		// next one. Order matters only in that both happen on the same scan -
		// the index clears OperationDone itself once it has seen it.
		FG_Transport.SetIndexOperationDone(Index := Index, Value := TRUE);
		Group.ChangeState(E_PMLCommand.ePMLCommand_Reset);

END_CASE

// Every other state - Execute, Starting, Resetting, Held, Aborted - is left
// alone on purpose. The index unit goes on waiting, and if the group never
// finishes, FB_TransferIndex raises its own fault 3 on the operation timeout.
// That is the intended report of a stuck group, and it belongs to the index unit
// rather than here.
END_METHOD

METHOD PROTECTED Clearing
VAR_INPUT
END_VAR
// A safety fault cannot be cleared while the safety fault is still present.
// This stalls in Clearing DELIBERATELY, which is why Clearing is one of the three
// states EnforceSafety excludes. Not a deadlock: it completes on its own the
// moment the mushroom is released or the last lock confirms, with no second press.
CASE SequenceState OF
	0:
		NoStateTasksToComplete := FALSE;
		SequenceState := SequenceState + 10;

	10:
		IF SafetyOk THEN
			StateTasksComplete := TRUE;
		END_IF
END_CASE

SUPER^.Clearing();
END_METHOD

METHOD PUBLIC CyclicLogic
VAR_INPUT
END_VAR
IF NOT _InitComplete THEN
	_InitComplete := Initialize();
	RETURN;
END_IF

// --- Cross-couplings between sibling equipment modules -----------------------
// Siblings never talk directly; the machine brokers what crosses between them.
// Evaluated EVERY SCAN: a handshake sampled once deadlocks.
// The laser gate permissive is no longer brokered here - the gates moved into
// FG_01, which reads its own limits.

// Evaluated before the state machine so a unit sees this scan's values.
BrokerIndexHandshakes();

// --- Infrastructure ---------------------------------------------------------
// Hand this module's own state and mode down to FG_System before the base walks
// its submodules, so the lock policy and the signal tower both act on this
// scan's values rather than last scan's.
FG_System.SetMachineIndication(State := _CurrentState, Mode := _CurrentMode);

EnforceSafety();

SUPER^.CyclicLogic();
END_METHOD

ACTION EnforceSafety:
// The whole safety layer, in one place.
// !! FUNCTIONAL DEMONSTRATION, NOT A SAFETY-RATED FUNCTION. A real cell puts
// guard interlocks and E-stops on TwinSAFE, never in standard PLC logic.
// Nothing here is rated, diagnosed or redundant.
//
// THE THREE EXCLUDED STATES ARE LOAD-BEARING - do not simplify them away:
//   Aborting / Aborted  re-issuing AbortImmediate() overwrites the operator's
//                       Clear on the scan it lands, so Aborted is never left.
//   Clearing            we are in Clearing BECAUSE safety broke; aborting out of
//                       it makes Clear impossible.
// Every other state aborts, Stopped and Resetting included.
//
// NO SCAN LAG: every input here is a getter over a located variable. Do NOT
// reuse FB_DigitalSensor for the mushrooms - it caches _Active inside its own
// CyclicLogic, which put the emergency stops one scan behind.
IF NOT SafetyOk
	AND	_CurrentState <> E_PMLState.ePMLState_Aborting
	AND	_CurrentState <> E_PMLState.ePMLState_Aborted
	AND	_CurrentState <> E_PMLState.ePMLState_Clearing THEN

	AbortImmediate();
END_IF
END_ACTION

METHOD PROTECTED FINAL Execute
VAR_INPUT
END_VAR
// The machine sequences its groups by hand here, so SUPER^.Execute() is
// deliberately not called - the base would drive the submodule state machine in
// parallel with this one.
// The groups are not sequenced here. Each is triggered by its own index unit
// through BrokerGroup; this method only keeps the ring running. Pallet order
// emerges from the physical chain, and several may be in the line at once.

CASE _CurrentMode OF

	//============================= PRODUCTION =================================
	E_PMLUnitMode.ePMLUnitMode_Production:

		// The transport ring runs continuously for as long as the machine is
		// producing, so it is started once and left in Execute.
		IF FG_Transport.CurrentState = E_PMLState.ePMLState_Idle THEN
			FG_Transport.ChangeState(E_PMLCommand.ePMLCommand_Start);
		END_IF

		// The functional groups are no longer free-run from here. Each one is
		// started by its own index unit, through BrokerIndexHandshakes, once that
		// unit has a pallet stopped and lifted - which is what the twin actually
		// specifies and what the free-run loop was standing in for.

	//======================= MAINTENANCE & MANUAL =============================
	E_PMLUnitMode.ePMLUnitMode_Maintenance, E_PMLUnitMode.ePMLUnitMode_Manual:
		;
END_CASE
END_METHOD

// The signal tower's flash phase, forwarded so MAIN can hand it to the panel
// control source and every flashing lamp on the machine blinks together.
PROPERTY PUBLIC IndicationFlash : BOOL
GET
IndicationFlash := FG_System.IndicationFlash;
END_GET
END_PROPERTY

METHOD PROTECTED Initialize : BOOL;
VAR
END_VAR
Initialize := FALSE;

CASE DescendantSequenceState OF
	0:
		// Registering is what makes the framework call a module's state methods.
		// An unregistered module never reaches Complete, so BrokerGroup takes its
		// "group is not there" branch and the index unit is silently bypassed - with
		// the group's I/O linked and its HMI tiles bound, which is what makes it look
		// finished. FG_01 shipped that way once.
		RegisterSubmodule(FG_Transport);
		RegisterSubmodule(FG_System);
		RegisterSubmodule(FG_01);
		RegisterSubmodule(FG_02);
		RegisterSubmodule(FG_03);
		RegisterSubmodule(FG_04);
		RegisterSubmodule(FG_05);

		_LogModeChanges		:= TRUE;
		_LogStateChanges	:= TRUE;
		DescendantSequenceState := DescendantSequenceState + 10;

	10:
		// The FG_01 gate permissive used to be forced TRUE here, because nothing
		// could read the real gate state. FG_Transport now owns those sensors and
		// publishes GatesClosed, so the stand-in is gone and the permissive is
		// driven cyclically in CyclicLogic instead - a one-shot here would latch
		// a stale value and defeat the interlock.
		DescendantSequenceState := DescendantSequenceState + 10;

	20:
		IF SUPER^.Initialize() THEN
			DescendantSequenceState := DescendantSequenceState + 10;
		END_IF

	30:
		Initialize := TRUE;
END_CASE
END_METHOD

// The machine's safety chain. Derived on every read, never stored.
// MODE IS THE GATE, and the two inputs are gated differently on purpose:
//   Emergency stops  EVERY mode. Manual is precisely the mode where somebody is
//                    inside the cell jogging a cylinder.
//   Guard doors      Production only. Maintenance and Manual are the only way
//                    into the cell, because the locks hold throughout Production.
// FG_System publishes the two facts and applies no policy: only this module owns
// the PackML mode.
PROPERTY PUBLIC SafetyOk : BOOL
GET
SafetyOk :=	NOT FG_System.EmergencyStopActive
			AND	(	(_CurrentMode <> E_PMLUnitMode.ePMLUnitMode_Production)
				OR	FG_System.GuardsSecure);
END_GET
END_PROPERTY

// THE FIVE PROCESS GROUPS ARE NOT STARTED BY THE MACHINE. This method exists to
// say so, and SUPER^.Starting() is deliberately not called.
// The base commands EVERY registered submodule to Start and will not leave
// Starting until all are in Execute - which ran all five station sequences on an
// empty line the moment Start was pressed. That is the bug this method fixes.
//
// The groups must still be REGISTERED: registration gets their CyclicLogic
// called, makes Undefined-vs-Idle meaningful to BrokerGroup, and carries Abort,
// Stop, Clear and Reset down from the states this method does not override.
//
// KNOWN LIMIT: Holding and Suspending are still the base implementations and gate
// on every submodule reaching Held/Suspended. A group parked in Idle rejects Hold
// and never gets there, so the machine would stall in Holding. Nothing commands
// Hold today. Adding a Hold button means overriding Holding/Unholding here on the
// same pattern: command only the submodules actually in Execute, and gate on those.
METHOD PROTECTED Starting
VAR_INPUT
END_VAR
// The two infrastructure groups do follow the machine into Execute. FG_Transport
// runs the ring for as long as the machine produces, and FG_System owns the
// signal tower and the door locks.
FG_System.ChangeState(E_PMLCommand.ePMLCommand_Start);
FG_Transport.ChangeState(E_PMLCommand.ePMLCommand_Start);

// Same completion gate as the base, over those two submodules only. The
// StateTasksComplete / NoStateTasksToComplete term is carried over unchanged so
// this method can grow its own step chain later without the gate going wrong.
IF FG_System.CurrentState = E_PMLState.ePMLState_Execute
	AND FG_Transport.CurrentState = E_PMLState.ePMLState_Execute
	AND (StateTasksComplete OR NoStateTasksToComplete) THEN

	NoStateTasksToComplete	:= TRUE;
	StateTasksComplete		:= FALSE;
	StateComplete();
END_IF
END_METHOD

END_FUNCTION_BLOCK

// ---- Modules/01 FG_System/FG_System.TcPOU
// FG_System - cell infrastructure: enclosure, six interlocked doors, two
// E-stops, signal tower. Processes no parts.
// It publishes GuardsSecure and EmergencyStopActive and applies NO policy to
// them - only Machine owns the PackML mode, so Machine composes SafetyOk.
// Contract: _workflow/reference/fg-system-safety.md
FUNCTION_BLOCK FG_System EXTENDS FB_PackML_BaseModule
VAR
	// Named exactly as the twin names them, so MAIN.Machine.FG_System.<name>
	// matches MAIN.FG_System.<name> in the twin's PLC tree. Side 1, then side 2.
	B_SafetyDoor11 : FB_SafetyDoor := (Name := 'B_SafetyDoor11');
	B_SafetyDoor12 : FB_SafetyDoor := (Name := 'B_SafetyDoor12');
	B_SafetyDoor13 : FB_SafetyDoor := (Name := 'B_SafetyDoor13');
	B_SafetyDoor21 : FB_SafetyDoor := (Name := 'B_SafetyDoor21');
	B_SafetyDoor22 : FB_SafetyDoor := (Name := 'B_SafetyDoor22');
	B_SafetyDoor23 : FB_SafetyDoor := (Name := 'B_SafetyDoor23');

	// One component per mushroom, signal bit and lamp bit together - they are one
	// device. Both read NORMALLY CLOSED: the input is TRUE while healthy, FALSE
	// while latched. Initialize sets .Inverted := TRUE for that, and SIM_1's
	// Mapping inverts the twin's FB_Button so the twin presents the same sense as
	// the real hardware. See _workflow/reference/plc-io-exceptions.md.
	SS_EStop1 : FB_IlluminatedButton := (Name := 'SS_EStop1');
	SS_EStop2 : FB_IlluminatedButton := (Name := 'SS_EStop2');

	H_SignalTower : FB_SignalTower := (Name := 'H_SignalTower');

	// Written by SetMachineIndication before this module's CyclicLogic runs.
	_MachineState : Tc3_PackML_V2.E_PMLState;
	_MachineMode : E_PMLUnitMode;

	_DoorsRequestedLocked : BOOL;

	{ attribute 'TcHmiSymbol.AddSymbol' }
	HMI : ST_HMI_FG_System;
END_VAR

METHOD PUBLIC CyclicLogic
VAR_INPUT
END_VAR
IF NOT _InitComplete THEN
	_InitComplete := Initialize();
	RETURN;
END_IF

// --- Lock policy ------------------------------------------------------------
// Sealed in Production, free in Maintenance and Manual. Commanded at power-up,
// so a reset never has to wait for a lock. Consequence: an operator in
// Production CANNOT open a door - getting in means selecting another mode.
_DoorsRequestedLocked := (_MachineMode = E_PMLUnitMode.ePMLUnitMode_Production);

B_SafetyDoor11.RequestLock := _DoorsRequestedLocked;
B_SafetyDoor12.RequestLock := _DoorsRequestedLocked;
B_SafetyDoor13.RequestLock := _DoorsRequestedLocked;
B_SafetyDoor21.RequestLock := _DoorsRequestedLocked;
B_SafetyDoor22.RequestLock := _DoorsRequestedLocked;
B_SafetyDoor23.RequestLock := _DoorsRequestedLocked;

// --- Indication -------------------------------------------------------------
// The tower shows the MACHINE's state, not this module's.
H_SignalTower.State := _MachineState;

// DriveEStopLamps runs BEFORE the base: FB_IlluminatedButton copies Lamp to its
// coil inside its own CyclicLogic, so setting Lamp after would be a scan late.
DriveEStopLamps();

// The base walks ipComponents, so everything set above is in place first.
SUPER^.CyclicLogic();

PublishStatus();
END_METHOD

ACTION DriveEStopLamps:
// dark = not latched, solid = latched, FLASHING = latched and machine Clearing.
// The flashing case says WHICH mushroom is blocking a clear, which solid-on-both
// cannot. Phase comes from the tower so everything blinks together.
// The decision lives here, not in FB_IlluminatedButton: a component must not
// know which PackML state the machine is in.
IF _MachineState = Tc3_PackML_V2.E_PMLState.ePMLState_Clearing THEN
	SS_EStop1.Lamp := SS_EStop1.Active AND H_SignalTower.Flash;
	SS_EStop2.Lamp := SS_EStop2.Active AND H_SignalTower.Flash;
ELSE
	SS_EStop1.Lamp := SS_EStop1.Active;
	SS_EStop2.Lamp := SS_EStop2.Active;
END_IF
END_ACTION

// TRUE while either mushroom is latched. Derived on every read.
// Machine acts on this in EVERY mode, unlike the guard doors.
PROPERTY EmergencyStopActive : BOOL
GET
EmergencyStopActive := SS_EStop1.Active OR SS_EStop2.Active;
END_GET
END_PROPERTY

// Every enclosure door shut AND locked. Closed alone is not enough.
// A getter, never a stored flag: a remembered readiness flag maintained in one
// state is stale in all the others.
PROPERTY GuardsSecure : BOOL
GET
GuardsSecure :=	B_SafetyDoor11.Secure
				AND	B_SafetyDoor12.Secure
				AND	B_SafetyDoor13.Secure
				AND	B_SafetyDoor21.Secure
				AND	B_SafetyDoor22.Secure
				AND	B_SafetyDoor23.Secure;
END_GET
END_PROPERTY

METHOD PROTECTED HMICommunication
VAR_INPUT
END_VAR
// Command half of the HMI bridge; PublishStatus is the status half. MUST be in
// this method: the base calls it immediately before ModeControl() and
// StateControl(), and reads its own PackMLBaseModule_HMI.Command, never ours.
PackMLBaseModule_HMI.Command := HMI.Command;

SUPER^.HMICommunication();

// The base clears a latch by writing back the value it acted on.
HMI.Command := PackMLBaseModule_HMI.Command;
END_METHOD

// The tower's flash phase, re-exposed so panel lamps blink with it rather than
// against it.
PROPERTY IndicationFlash : BOOL
GET
IndicationFlash := H_SignalTower.Flash;
END_GET
END_PROPERTY

METHOD PROTECTED Initialize : BOOL;
VAR
END_VAR
Initialize := FALSE;

CASE DescendantSequenceState OF
	0:
		// Nine components. Forgetting one is SILENT: its CyclicLogic is never
			// called, and the device reports nothing for ever.
		RegisterComponent(B_SafetyDoor11);
		RegisterComponent(B_SafetyDoor12);
		RegisterComponent(B_SafetyDoor13);
		RegisterComponent(B_SafetyDoor21);
		RegisterComponent(B_SafetyDoor22);
		RegisterComponent(B_SafetyDoor23);
		RegisterComponent(SS_EStop1);
		RegisterComponent(SS_EStop2);
		RegisterComponent(H_SignalTower);

		// NC sense, and it belongs in step 0 rather than with the other parameters
		// in step 10: Machine.EnforceSafety reads EmergencyStopActive through a
		// getter that does not care whether this module has initialised, so every
		// scan the polarity is still FALSE is a scan a healthy mushroom reads as
		// LATCHED and aborts the machine. Set it in the same step that registers
		// the components, and there is no such scan after the first.
		//
		// The process-image bit is TRUE while the mushroom is HEALTHY and FALSE
		// while latched - a real normally-closed contact, and what SIM_1's Mapping
		// now emits. Active is HardwareInput XOR _Inverted, so Active stays TRUE
		// while pressed and EmergencyStopActive is unchanged.
		//
		// With no process image at all - SIM_1 not running, EtherCAT down, a cut
		// cable - both bits read 0, so both mushrooms report ACTIVE and the machine
		// will not leave Aborted. That is the fail-safe direction and it is
		// intended. See _workflow/reference/plc-io-exceptions.md.
		SS_EStop1.Inverted := TRUE;
		SS_EStop2.Inverted := TRUE;

		_LogModeChanges		:= FALSE;
		_LogStateChanges	:= TRUE;
		DescendantSequenceState := DescendantSequenceState + 10;

	10:
		// A lock has 3 s to confirm before its door raises fault 1.
		B_SafetyDoor11.LockTime := T#3S;
		B_SafetyDoor12.LockTime := T#3S;
		B_SafetyDoor13.LockTime := T#3S;
		B_SafetyDoor21.LockTime := T#3S;
		B_SafetyDoor22.LockTime := T#3S;
		B_SafetyDoor23.LockTime := T#3S;

		H_SignalTower.FlashTime := T#500MS;

		DescendantSequenceState := DescendantSequenceState + 10;

	20:
		IF SUPER^.Initialize() THEN
			DescendantSequenceState := DescendantSequenceState + 10;
		END_IF

	30:
		Initialize := TRUE;
END_CASE
END_METHOD

ACTION PublishStatus:
// Status half of the HMI bridge. Called AFTER SUPER^.CyclicLogic(), so every
// field is this scan's.
HMI.Config	:= PackMLBaseModule_HMI.Config;
HMI.Status	:= PackMLBaseModule_HMI.Status;

HMI.StateName := F_PMLStateName(_CurrentState);

// --- Safety -----------------------------------------------------------------
HMI.Safety.GuardsSecure			:= GuardsSecure;
HMI.Safety.EmergencyStopActive	:= EmergencyStopActive;
HMI.Safety.DoorsRequestedLocked	:= _DoorsRequestedLocked;

HMI.Safety.DoorClosed[1] := B_SafetyDoor11.Closed;
HMI.Safety.DoorClosed[2] := B_SafetyDoor12.Closed;
HMI.Safety.DoorClosed[3] := B_SafetyDoor13.Closed;
HMI.Safety.DoorClosed[4] := B_SafetyDoor21.Closed;
HMI.Safety.DoorClosed[5] := B_SafetyDoor22.Closed;
HMI.Safety.DoorClosed[6] := B_SafetyDoor23.Closed;

HMI.Safety.DoorLocked[1] := B_SafetyDoor11.Locked;
HMI.Safety.DoorLocked[2] := B_SafetyDoor12.Locked;
HMI.Safety.DoorLocked[3] := B_SafetyDoor13.Locked;
HMI.Safety.DoorLocked[4] := B_SafetyDoor21.Locked;
HMI.Safety.DoorLocked[5] := B_SafetyDoor22.Locked;
HMI.Safety.DoorLocked[6] := B_SafetyDoor23.Locked;

HMI.Safety.DoorFaultCode[1] := B_SafetyDoor11.FaultCode;
HMI.Safety.DoorFaultCode[2] := B_SafetyDoor12.FaultCode;
HMI.Safety.DoorFaultCode[3] := B_SafetyDoor13.FaultCode;
HMI.Safety.DoorFaultCode[4] := B_SafetyDoor21.FaultCode;
HMI.Safety.DoorFaultCode[5] := B_SafetyDoor22.FaultCode;
HMI.Safety.DoorFaultCode[6] := B_SafetyDoor23.FaultCode;

HMI.Safety.EStopActive[1] := SS_EStop1.Active;
HMI.Safety.EStopActive[2] := SS_EStop2.Active;
END_ACTION

// The machine hands its state and mode down every scan. A parent commanding its
// direct child is the only direction SPT layering allows.
// MUST be called before the machine's SUPER^.CyclicLogic(), which is what calls
// this module's CyclicLogic - otherwise both act on last scan's state.
METHOD PUBLIC SetMachineIndication
VAR_INPUT
	State : Tc3_PackML_V2.E_PMLState;
	Mode : E_PMLUnitMode;
END_VAR
_MachineState	:= State;
_MachineMode	:= Mode;
END_METHOD

END_FUNCTION_BLOCK

// ---- Library/POUs/FB_SafetyDoor.TcPOU
// ============================================================================
// One interlocked enclosure door with a safety lock. Maps to the twin's FB_Lock:
// bClosed and bLocked come back as two channels, bLock goes out as one coil.
//
// AN OPEN DOOR IS NOT A FAULT OF THIS COMPONENT - it is simply Closed = FALSE,
// which the owning module folds into GuardsSecure. _Error is raised only by a
// genuine device failure (a lock commanded and never confirmed), because the SPT
// base waits on every component's Error in Clearing: raising it for a door somebody
// deliberately opened would stall Clearing in Maintenance, where the whole point is
// that safety is ignored.
FUNCTION_BLOCK FB_SafetyDoor EXTENDS FB_ComponentBase
VAR
	ClosedSensor AT %I* : BOOL;
	LockedSensor AT %I* : BOOL;
	LockOutput AT %Q* : BOOL;

	_RequestLock : BOOL;
	_FaultCode : UDINT;
	_LockTime : TIME := T#3S;
	LockTimer : TON;

	// Safety door - closed, locked, and the lock fault
	{ attribute 'TcHmiSymbol.AddSymbol' }
	HMI : ST_SafetyDoor_HMI;
END_VAR

// TRUE while the door leaf is shut. Says nothing about the lock.
PROPERTY Closed : BOOL
GET
Closed := ClosedSensor;
END_GET
END_PROPERTY

METHOD PUBLIC CyclicLogic
VAR_INPUT
END_VAR
IF NOT _InitComplete THEN
	_InitComplete := Initialize();
	RETURN;
END_IF

// The coil follows the request unconditionally. A lock fault must never drop the
// lock - that would open the cell in response to a failure to close it.
LockOutput := _RequestLock;

// Fault 1: lock commanded and never confirmed. Re-raises for as long as the
// physical condition lasts, the same shape FB_AbstractBinaryDrive uses for its
// drive-not-active fault.
LockTimer(IN := LockOutput AND NOT LockedSensor, PT := _LockTime);
IF LockTimer.Q THEN
	_FaultCode := 1;
END_IF

_Busy		:= LockOutput AND NOT LockedSensor;
_Error		:= _FaultCode <> 0;
_ErrorID	:= _FaultCode;

SUPER^.CyclicLogic();

// Device config and status only; the inherited half is bridged in
// HMICommunication. Publishing is not filling - without these the struct would be
// a live ADS symbol reading zeros, and a panel would show six doors that are
// neither closed nor locked whatever the cell is doing.
HMI.DeviceConfig.LockTime		:= _LockTime;
HMI.Device.Closed				:= ClosedSensor;
HMI.Device.Locked				:= LockedSensor;
HMI.Device.Secure				:= ClosedSensor AND LockedSensor;
HMI.Device.LockRequested		:= _RequestLock;
HMI.Device.FaultCode			:= _FaultCode;
END_METHOD

METHOD PROTECTED HMICommunication
VAR_INPUT
END_VAR
// HMI is a published mirror of the base's own ComponentBase_HMI - carry operator
// intent in before the base looks, and its answers back out afterwards.
//
// The inherited Command.Reset is the one writable member that matters here: it is
// how an operator clears fault 1 once a sticky lock has been dealt with.
ComponentBase_HMI.Command := HMI.Command;

SUPER^.HMICommunication();

HMI.Config	:= ComponentBase_HMI.Config;
HMI.Status	:= ComponentBase_HMI.Status;
HMI.Command	:= ComponentBase_HMI.Command;

// A zero lock time would make the fault fire on the scan the lock is commanded,
// before any real lock could answer, so it is refused rather than obeyed.
IF HMI.DeviceConfig.LockTime > T#0S THEN
	_LockTime := HMI.DeviceConfig.LockTime;
END_IF
END_METHOD

// 0 none, 1 lock commanded but never confirmed.
PROPERTY FaultCode : UDINT
GET
FaultCode := _FaultCode;
END_GET
END_PROPERTY

METHOD PROTECTED Initialize : BOOL
VAR_INPUT
END_VAR
Initialize := SUPER^.Initialize();
END_METHOD

// How long the lock has to confirm before fault 1 is raised.
PROPERTY LockTime : TIME
GET
LockTime := _LockTime;
END_GET
SET
_LockTime := LockTime;
END_SET
END_PROPERTY

// TRUE while the lock reports engaged.
PROPERTY Locked : BOOL
GET
Locked := LockedSensor;
END_GET
END_PROPERTY

// Written every scan by the owning module from the machine's PackML mode.
PROPERTY RequestLock : BOOL
GET
RequestLock := _RequestLock;
END_GET
SET
_RequestLock := RequestLock;
END_SET
END_PROPERTY

METHOD PUBLIC Reset : BOOL
VAR_INPUT
END_VAR
Reset := SUPER^.Reset();
IF Reset THEN
	_FaultCode := 0;
END_IF
END_METHOD

// The whole safety contribution of this door: shut AND locked. Derived on every
// read, never stored - a remembered readiness flag is what put two pallets on one
// lift carriage, see transport-behaviour.md.
PROPERTY Secure : BOOL
GET
Secure := ClosedSensor AND LockedSensor;
END_GET
END_PROPERTY

END_FUNCTION_BLOCK

// ---- Library/POUs/FB_IlluminatedButton.TcPOU
// ============================================================================
// A button that reports and lights: one input bit, one output bit, one device.
// Maps to the twin's OC_Core FB_Button - bValue (0 released, 1 pressed) and
// bEnable (0 lamp off, 1 lamp on), verified against the OC_Core 1.3.1 binary.
//
// Active IS A LIVE GETTER over the located input, not a cached value. That is why
// this exists instead of FB_DigitalSensor, which computes _Active inside its own
// CyclicLogic and so put a ONE-SCAN LAG on the emergency stops in
// Machine.EnforceSafety. No debounce, no simulation, no timers.
//
// LAYERING: this component does not know what a PackML state is, so it does not
// decide whether its lamp is solid or flashing. It exposes Lamp; the owning module
// writes it - see FG_System.DriveEStopLamps.
//
// !! NOT A SAFETY-RATED COMPONENT. A real emergency stop belongs on TwinSAFE.
FUNCTION_BLOCK FB_IlluminatedButton EXTENDS FB_ComponentBase
VAR
	HardwareInput AT %I* : BOOL;
	LampOutput AT %Q* : BOOL;

	_Lamp : BOOL;
	_Inverted : BOOL;

	// Illuminated button - pressed state, lamp and contact polarity
	{ attribute 'TcHmiSymbol.AddSymbol' }
	HMI : ST_IlluminatedButton_HMI;
END_VAR

// TRUE while the button is pressed. Read straight off the located input, so it is
// this scan's value no matter when the caller reads it - see the header.
PROPERTY Active : BOOL
GET
Active := HardwareInput XOR _Inverted;
END_GET
END_PROPERTY

METHOD PUBLIC CyclicLogic
VAR_INPUT
END_VAR
IF NOT _InitComplete THEN
	_InitComplete := Initialize();
	RETURN;
END_IF

// The whole of it. Active needs no work here - it is a getter over the input.
LampOutput := _Lamp;

_Busy	:= FALSE;
_Error	:= FALSE;

SUPER^.CyclicLogic();

// Device config and status only. The inherited Config / Command / Status half of
// HMI mirrors ComponentBase_HMI and is bridged in HMICommunication.
//
// Publishing is not filling: without these four lines the struct would be a live
// ADS symbol reading zeros forever, which on a panel looks exactly like a button
// nobody is pressing.
HMI.DeviceConfig.Inverted	:= _Inverted;
HMI.Device.Active			:= HardwareInput XOR _Inverted;
HMI.Device.Lamp				:= LampOutput;
END_METHOD

METHOD PROTECTED HMICommunication
VAR_INPUT
END_VAR
// HMI is a published mirror of the base's own ComponentBase_HMI - carry operator
// intent in before the base looks, and its answers back out afterwards. Same
// shape as FB_AbstractBinaryDrive.
ComponentBase_HMI.Command := HMI.Command;

SUPER^.HMICommunication();

HMI.Config	:= ComponentBase_HMI.Config;
HMI.Status	:= ComponentBase_HMI.Status;
HMI.Command	:= ComponentBase_HMI.Command;

// Polarity is commissioning configuration, so the panel may set it - but only
// while the PLC says HMI control is available for this component.
IF ComponentBase_HMI.Status.HMIControlAvailable THEN
	_Inverted := HMI.DeviceConfig.Inverted;
END_IF
END_METHOD

METHOD PROTECTED Initialize : BOOL
VAR_INPUT
END_VAR
// Seed the HMI mirror from the configured polarity BEFORE anything can read it
// back. HMICommunication assigns _Inverted := HMI.DeviceConfig.Inverted whenever
// HMI control is available, and CyclicLogic only publishes the other direction
// AFTER SUPER^.CyclicLogic() has already called it - so on the first executing
// scan the mirror is still the struct's zero default. Without this line, a
// polarity set by the owning module would be silently reverted to FALSE the
// moment the machine was in Manual, which on an emergency stop is the failure
// that matters. Idempotent: Initialize runs every scan until it returns TRUE.
HMI.DeviceConfig.Inverted := _Inverted;

Initialize := SUPER^.Initialize();
END_METHOD

// Input polarity of the contact. TRUE means the input is NORMALLY CLOSED: it
// reads TRUE while healthy and FALSE while pressed, so Active is the inverse.
//
// THE TWO EMERGENCY STOPS SET THIS TRUE, in FG_System.Initialize. A physical
// mushroom is wired normally-closed, and the failure mode of getting it the
// other way round is the worst one there is: a cut cable would read as "no
// emergency stop". SIM_1's Mapping inverts the twin's FB_Button - which reports
// bValue TRUE while PRESSED - so the twin presents that same NC sense and the
// control program does not change between twin and hardware.
// See _workflow/reference/plc-io-exceptions.md.
PROPERTY Inverted : BOOL
GET
Inverted := _Inverted;
END_GET
SET
_Inverted := Inverted;
END_SET
END_PROPERTY

// The lamp request. Written every scan by the owning module, which is the only
// level that knows whether this should be solid, flashing or dark.
PROPERTY Lamp : BOOL
GET
Lamp := _Lamp;
END_GET
SET
_Lamp := Lamp;
END_SET
END_PROPERTY

END_FUNCTION_BLOCK

// ---- Library/POUs/FB_SignalTower.TcPOU
// ============================================================================
// Four colour signal tower, driven from the machine's PackML state.
// Implements _workflow/reference/state-lamp.md. Two things that page is misread on:
//   1. the rows are INDEPENDENT CONDITIONS, not a priority ladder - two lamps can
//      legitimately be lit at once;
//   2. its "Completed" column is V4 spelling. This project runs SPT V3.9, where the
//      state is ePMLState_Complete and ePMLState_Completed will not compile.
//
// Amber and blue have no source in this machine yet - the inputs are present,
// default FALSE and never asserted, so the table can be completed later without
// touching the lamp logic. There is no horn device in the twin.
//
// State is written every scan by the owning module with the MACHINE's state, not
// FG_System's own: Machine.Execute deliberately does not call SUPER^.Execute(), so
// a tower driven from its own module would sit dark all through production.
FUNCTION_BLOCK FB_SignalTower EXTENDS FB_ComponentBase
VAR
	Red AT %Q* : BOOL;
	Yellow AT %Q* : BOOL;
	Blue AT %Q* : BOOL;
	Green AT %Q* : BOOL;

	_State : Tc3_PackML_V2.E_PMLState;

